// TIA Portal project "Madeta" (V14)

(* hardware
DEVICE "ET 200S station_1"  ET 200S station
   slot 0: "Rack_0"  Rail
   slot 2: "PLC Paletizace pytlu"  IM 151-8 PN/DP CPU  6ES7 151-8AB01-0AB0  V3.2
      slot 1: "PROFINET interface_1"  PN-IO
         slot 1: "Port_1"  Port
         slot 2: "Port_2"  Port
         slot 3: "Port_3"  Port
   slot 4: "PM-E 24VDC_1"  PM-E 24VDC  6ES7 138-4CA01-0AA0
   slot 5: "8DI x 24VDC_1"  8DI x 24VDC  6ES7 131-4BF00-0AA0
   slot 6: "8DI x 24VDC_2"  8DI x 24VDC  6ES7 131-4BF00-0AA0
   slot 7: "8DI x 24VDC_3"  8DI x 24VDC  6ES7 131-4BF00-0AA0
   slot 8: "8DI x 24VDC_4"  8DI x 24VDC  6ES7 131-4BF00-0AA0
   slot 9: "8DI x 24VDC_5"  8DI x 24VDC  6ES7 131-4BF00-0AA0
   slot 10: "8DI x 24VDC_6"  8DI x 24VDC  6ES7 131-4BF00-0AA0
   slot 11: "PM-E 24VDC_2"  PM-E 24VDC  6ES7 138-4CA01-0AA0
   slot 12: "8DO x 24VDC / 0.5A_1"  8DO x 24VDC / 0.5A  6ES7 132-4BF00-0AA0
   slot 13: "PM-E 24VDC_3"  PM-E 24VDC  6ES7 138-4CA01-0AA0
   slot 14: "8DO x 24VDC / 0.5A_2"  8DO x 24VDC / 0.5A  6ES7 132-4BF00-0AA0
   slot 15: "8DO x 24VDC / 0.5A_3"  8DO x 24VDC / 0.5A  6ES7 132-4BF00-0AA0
   slot 16: "8DO x 24VDC / 0.5A_4"  8DO x 24VDC / 0.5A  6ES7 132-4BF00-0AA0
   slot 17: "8DO x 24VDC / 0.5A_5"  8DO x 24VDC / 0.5A  6ES7 132-4BF00-0AA0
DEVICE "GSD device_1"  GSD.Device.PN
   slot 0: "Rack"  Rack  V1.0
   slot 0: "COMAU PAL 180"  X20IF10E3-1  X20IF10E3-1  2.1.x
      slot 0: "DIM 1"  DIM 1
      slot 1: "Interface"  Interface
         slot 1: "Interface - Port1"  Interface - Port1
         slot 2: "Interface - Port2"  Interface - Port2
   slot 1: "8 Bytes In_1"  8 Bytes In
      slot 0: "9"  9
   slot 2: "8 Bytes Out_1"  8 Bytes Out
      slot 0: "10"  10
DEVICE "Panel paletizace pytlu"  KTP600 Basic color PN
   slot 0: "KTP600 Basic color PN"  KTP600 Basic color PN  6AV6 647-0AD11-3AX0  12.0.0.0
   slot 1: "HMI_RT_2"  KTP600 Basic color PN  6AV6 647-0AD11-3AX0  12.0.0.0
   slot 5: "Panel paletizace pytlu.IE_CP_1"  PROFINET Interface  12.0.0.0
      slot 1: "PROFINET Interface_1"  PROFINET Interface
         slot 1: "Port_1"  Port
*)

// ===== PLC "PLC Paletizace pytlu"  IM 151-8 PN/DP CPU =====

VAR_GLOBAL   // PLC tag table "Default tag table"
   "Tag_1" AT %M50.0 : Bool;
   "Manual_Dopravnik_P1" AT %M50.1 : Bool;
   "Manual_Dopravnik_P2_k _oviječce" AT %M50.2 : Bool;
   "Manual_Dopravnik_P3" AT %M50.3 : Bool;
   "Manual_PaletaRovnani_Rozevrit" AT %M60.0 : Bool;
   "Manual_PaletaRovnani_Sevrit" AT %M60.2 : Bool;
   "Manual_Zarazka_P2_Dolu" AT %M60.3 : Bool;
   "Manual_Zarazka_P2_Nahoru" AT %M60.4 : Bool;
   "Manual_Valcovacka" AT %M60.5 : Bool;
   "Automat" AT %M100.0 : Bool;
   "Dopravnik P1 Start" AT %Q6.0 : Bool;
   "Dopravnik P2 do Ovíječky" AT %Q6.1 : Bool;
   "Dopravnik P3 Start" AT %Q6.2 : Bool;
   "Valcovacka Start" AT %Q6.7 : Bool;
   "PaletaRovnani_Rozevrit" AT %Q6.3 : Bool;
   "PaletaRovnani_Sevrit" AT %Q6.4 : Bool;
   "Dopravnik P2 do Stohu" AT %Q6.6 : Bool;
   "Zarazka_P2_Dolu" AT %Q6.5 : Bool;
   "Dveře 2 otevřit" AT %Q7.0 : Bool;
   "Dveře 1 otevřit" AT %Q7.2 : Bool;
   "Dveře 1 otevřeno" AT %Q7.1 : Bool;
   "Dveře 2 otevřeno" AT %Q7.3 : Bool;
   "Dveře 1 požadavek" AT %I3.2 : Bool;
   "Dveře 2 požadavek" AT %I3.5 : Bool;
   "Signální sloupek zelená" AT %Q9.4 : Bool;
   "Tag_2" AT %M150.4 : Bool;
   "Optická závora override" AT %Q10.0 : Bool;
   "Reset" AT %I0.5 : Bool;
   "Override" AT %I0.6 : Bool;
   "Optická závora zapnutí" AT %Q10.1 : Bool;
   "Error" AT %M101.0 : Bool;
   "OP_Start" AT %M90.0 : Bool;
   "OP_Stop" AT %M90.1 : Bool;
   "Tag_3" AT %M200.0 : Bool;
   "Tag_4" AT %M120.0 : Bool;
   "Tag_5" AT %M200.1 : Bool;
   "PřesunP2naOvijecka" AT %M220.0 : Bool;
   "PřesunOvijeckanaP3" AT %M220.1 : Bool;
   "Manual_Oviječka" AT %M50.4 : Bool;
   "Dopravnik Ovijecka Start" AT %Q7.7 : Bool;
   "Manual_Váha" AT %M60.6 : Bool;
   "Pytel na P1" AT %I4.0 : Bool;
   "Rovnání P2 otevřeno" AT %I4.2 : Bool;
   "Paleta P2 u Ovíječky" AT %I4.4 : Bool;
   "Srovnaná paleta na P2" AT %T50 : Timer;
   "Volno na P3" AT %I4.5 : Bool;
   "Ovíječka_Konec balení" AT %I2.5 : Bool;
   "Komunikace robot byte 1" AT %QB256 : Byte;
   "Časovač vypínací impulz váha dopravník" AT %T122 : Timer;
   "Ovíječka_Volná trať" AT %I2.4 : Bool;
   "Ovíječka_Porucha" AT %I2.6 : Bool;
   "Ovíječka_Paleta na točně" AT %I2.7 : Bool;
   "Ovíječce_Start balení" AT %Q9.0 : Bool;
   "Ovíječce_Možno balit" AT %Q9.1 : Bool;
   "Ovíječka_Povolení otevřít dveře" AT %I1.3 : Bool;
   "Manual_RučníPřesunOvnaP3" AT %M50.5 : Bool;
   "Manual_RučníPřesunP2naOv" AT %M50.6 : Bool;
   "Nouzové zastavení" AT %I0.2 : Bool;
   "Tag_6" AT %M200.2 : Bool;
   "Tag_7" AT %T60 : Timer;
   "Pytel na konci Válcovačky" AT %I4.6 : Bool;
   "Časovač volno na váze" AT %T61 : Timer;
   "Tag_9" AT %T62 : Timer;
   "Paleta P2 u stohu" AT %I4.3 : Bool;
   "Manual_Dopravnik_P2_ke_stohu" AT %M50.7 : Bool;
   "Manual_Paletu_P2_ke_stohu" AT %M51.0 : Bool;
   "Manual_Paletu_P2_k_ovíječce" AT %M51.1 : Bool;
   "Časovač_paleta u stohu" AT %T63 : Timer;
   "Časovač_paleta u ovíječky" AT %T64 : Timer;
   "Časovač paleta v ovíječce" AT %T65 : Timer;
   "Timer" AT %T80 : Timer;
   "PHrana I258.4" AT %M80.0 : Bool;
   "Časovač_zapni_pohon_robota" AT %T81 : Timer;
   "Zařízení zapnuto" AT %I0.3 : Bool;
   "Časovač_zapni automat robota" AT %T82 : Timer;
   "Časovač_vypnutí automatu robota" AT %T83 : Timer;
   "Časovač_vypnutí pohonů robota" AT %T84 : Timer;
   "Časovač_spoždění_zapnutí_pohonů robota" AT %T85 : Timer;
   "Časovač_reset alarmů robota" AT %T86 : Timer;
   "Časovač_zpoždění startu" AT %T87 : Timer;
   "Přítomnost palety P2" AT %I4.1 : Bool;
   "Časovač_váha volná" AT %T59 : Timer;
   "Jistič dopravníku P1,P2" AT %I0.1 : Bool;
   "Časovač vadný pytel na váze" AT %T58 : Timer;
   "volný" AT %T123 : Timer;
   "Časovač_start balení" AT %T66 : Timer;
   "Dveře 1 potvrzeno zavření" AT %I3.1 : Bool;
   "Dveře 2 potvrzeno zavření" AT %I3.4 : Bool;
   "Nízký tlak vzduchu" AT %I0.4 : Bool;
   "Jistič válcovačky nebo dopravníku ovíječky" AT %I0.7 : Bool;
   "Porucha kontaktů bezpečnostního relé" AT %I1.0 : Bool;
   "Časovač příliš dlouhý přesun z dopravníku P2" AT %T90 : Timer;
   "Časovač příliš dlouhý přesun z ovíječky" AT %T91 : Timer;
   "Časovač příliš dlouhý přesun palety na dopravníku P2 k ovíječce" AT %T92 : Timer;
   "Časovač píliš dlouhý přesun palety na dopravníku P2 ke stohu" AT %T93 : Timer;
   "Časovač příliš dlouhý chod rovnání palety k paletě" AT %T94 : Timer;
   "Časovač příliš dlouhý chod rovnání palety od palety" AT %T95 : Timer;
   "Světelná závora OK" AT %I1.2 : Bool;
   "Časovač volno na P3" AT %T68 : Timer;
   "Robotovi paleta ve stohu připravena" AT %Q259.0 : Bool;
   "Časovač nová paleta na zmetky" AT %T88 : Timer;
   "Časovač impuls nová paleta na zmetky" AT %T99 : Timer;
   "Signální  sloupek červená" AT %Q9.6 : Bool;
   "Signální sloupek houkačka" AT %Q9.7 : Bool;
   "Signální sloupek oranžová" AT %Q9.5 : Bool;
   "Tag_12" AT %M110.0 : Bool;
   "Tag_13" AT %M110.1 : Bool;
   "Tag_14" AT %M110.2 : Bool;
   "Tag_15" AT %M110.3 : Bool;
   "Tag_8" AT %M150.3 : Bool;
   "Tag_11" AT %M150.0 : Bool;
   "Tag_16" AT %M150.7 : Bool;
   "Tag_17" AT %M150.2 : Bool;
   "Dveře 1 otevřeny" AT %I3.3 : Bool;
   "Tag_18" AT %M40.0 : Bool;
   "Signální sloupek modrá" AT %Q8.7 : Bool;
   "Nouzové zastavení robot neaktivní" AT %I3.6 : Bool;
   "Nouzové zastavení ovíječka neaktivní" AT %I3.7 : Bool;
   "Dveře 2 otevřeny" AT %I3.0 : Bool;
END_VAR

VAR_GLOBAL   // PLC tag table "Errors"
   "Jistič dopravníku P1" AT %I0.0 : Bool;
END_VAR

VAR_GLOBAL   // PLC tag table "Komunikace_robot"
   "Robot_Paletu do pozice stoh" AT %I258.1 : Bool;
   "Robot_paletu do pozice u ovíječky" AT %I258.2 : Bool;
   "Robotovi_P1_Paleta_u_stohu" AT %Q258.0 : Bool;
   "Robotovi_P2_Paleta_u_ovíječky" AT %Q258.1 : Bool;
   "Robotovi_Vadný_pytel" AT %Q258.2 : Bool;
   "Robotovi_Pytel_na_dopravníku" AT %Q258.3 : Bool;
   "Robotovi_polož_novou_paletu" AT %Q258.4 : Bool;
   "Robotovi_paleta_na_zmetky_připravena" AT %Q258.5 : Bool;
   "Robotovi_start_produkce" AT %Q258.6 : Bool;
   "Robotovi_konec_produkce" AT %Q258.7 : Bool;
   "Robotovi_artikl" AT %QB260 : Byte;
   "Robotovi_max_počet_vrstev" AT %QB261 : Byte;
   "Robotovi_aktualní_počet_vrstev" AT %QB262 : Byte;
   "Robotovi_aktualní_počet_pytlů" AT %QB263 : Byte;
   "Robot_potvrzení_zmetku" AT %I258.3 : Bool;
   "Robot_pytel_položen" AT %I258.4 : Bool;
   "Robot_nová_paleta_položena" AT %I258.5 : Bool;
   "Robot_jsem_mimo_dopravník_P1" AT %I258.6 : Bool;
   "Robot_paleta_vadných_polovina" AT %I258.7 : Bool;
   "Robot_paleta_vadných_plná" AT %I259.0 : Bool;
   "Robot_mimo_paletu" AT %I259.1 : Bool;
   "Robot_paleta_plná" AT %I259.2 : Bool;
   "Robot_No alarm" AT %I256.0 : Bool;
   "Robot_Drive on status" AT %I256.1 : Bool;
   "Robot_Start / no hold on mot prog" AT %I256.2 : Bool;
   "Robot_Remote" AT %I256.3 : Bool;
   "Robot_Teach enable (DRI.ON+T1)" AT %I256.4 : Bool;
   "Robot_U1" AT %I256.5 : Bool;
   "Robot_U2" AT %I256.6 : Bool;
   "Robot_U3" AT %I256.7 : Bool;
   "Robot_U4" AT %I257.0 : Bool;
   "Robot_No activa latch alarm" AT %I257.1 : Bool;
   "Robot_Safety speed (for remote)" AT %I257.2 : Bool;
   "Robot_Programing mode" AT %I257.3 : Bool;
   "Robot_State selector in local or remote" AT %I257.5 : Bool;
   "Robot_Systém reddy" AT %I257.6 : Bool;
   "Robot_Heart bit" AT %I257.7 : Bool;
   "Robot_is on HOME" AT %I258.0 : Bool;
   "Robot_reserve" AT %I257.4 : Bool;
   "Robotovi_Drive ON" AT %Q256.0 : Bool;
   "Robotovi_No drive OFF" AT %Q256.1 : Bool;
   "Robotovi_Start" AT %Q256.2 : Bool;
   "Robotovi_No hold" AT %Q256.3 : Bool;
   "Robotovi_U1" AT %Q256.4 : Bool;
   "Robotovi_U2" AT %Q256.5 : Bool;
   "Robotovi_U3" AT %Q256.6 : Bool;
   "Robotovi_U4" AT %Q256.7 : Bool;
   "Robotovi_Cancel alarm" AT %Q257.0 : Bool;
   "Robotovi_Safety speed" AT %Q257.1 : Bool;
   "Robotovi_Reserve" AT %Q257.2 : Bool;
   "Robotovi_Reserve_1" AT %Q257.3 : Bool;
   "Robotovi_Reserve_2" AT %Q257.4 : Bool;
   "Robotovi_Reserve_3" AT %Q257.5 : Bool;
   "Robotovi_Reserve_4" AT %Q257.6 : Bool;
   "Robotovi_Reserve_5" AT %Q257.7 : Bool;
END_VAR

VAR_GLOBAL   // PLC tag table "Komunikace_váha"
   "Váha_Nouzové zastavení" AT %I2.1 : Bool;
   "Váha_Snímač na dopravníku volno" AT %I2.3 : Bool;
   "Dopravník Váha Start" AT %Q8.4 : Bool;
   "Dopravník Váha Stop" AT %Q8.5 : Bool;
   "Váha_motory_zapnuty" AT %I2.0 : Bool;
   "Váha_hmotnost_OK" AT %I2.2 : Bool;
END_VAR

TYPE "Karton"
   STRUCT
      Rotace : Bool;
      Pořadí : Int;
   END_STRUCT;
END_TYPE

// folder: DB

DATA_BLOCK "Komunikace vaha_DB"   // DB3
{ S7_Optimized_Access := 'FALSE' }
VERSION : 0.1
// stored: InstanceOfName Komunikace vaha
"Komunikace vaha"
BEGIN
END_DATA_BLOCK

DATA_BLOCK "Počítadlo_DB"   // DB5
{ S7_Optimized_Access := 'FALSE' }
VERSION : 0.1
// stored: InstanceOfName Počítadlo
"Počítadlo"
BEGIN
END_DATA_BLOCK

DATA_BLOCK "Dopravniky_DB"   // DB10
{ S7_Optimized_Access := 'FALSE' }
VERSION : 0.1
// stored: InstanceOfName Dopravniky
"Dopravniky"
BEGIN
END_DATA_BLOCK

DATA_BLOCK "Klapky_DB"   // DB11
{ S7_Optimized_Access := 'FALSE' }
VERSION : 0.1
// stored: InstanceOfName Klapky
"Klapky"
BEGIN
END_DATA_BLOCK

DATA_BLOCK "Dopravníky pytlů_DB"   // DB12
{ S7_Optimized_Access := 'FALSE' }
VERSION : 0.1
// stored: InstanceOfName Dopravníky pytlů
"Dopravníky pytlů"
BEGIN
END_DATA_BLOCK

DATA_BLOCK "Komunikace robot_DB"   // DB51
{ S7_Optimized_Access := 'FALSE' }
VERSION : 0.1
// stored: InstanceOfName Komunikace robot
"Komunikace robot"
BEGIN
END_DATA_BLOCK

DATA_BLOCK "Komunikace ovijecka_DB"   // DB52
{ S7_Optimized_Access := 'FALSE' }
VERSION : 0.1
// stored: InstanceOfName Komunikace ovijecka
"Komunikace ovijecka"
BEGIN
END_DATA_BLOCK

DATA_BLOCK "Opticka zavora_DB"   // DB54
{ S7_Optimized_Access := 'FALSE' }
VERSION : 0.1
// stored: InstanceOfName Opticka zavora
"Opticka zavora"
BEGIN
END_DATA_BLOCK

DATA_BLOCK "Dvere_DB"   // DB60
{ S7_Optimized_Access := 'FALSE' }
VERSION : 0.1
// stored: InstanceOfName Dvere
"Dvere"
BEGIN
END_DATA_BLOCK

DATA_BLOCK "Signalni sloupek_DB"   // DB61
{ S7_Optimized_Access := 'FALSE' }
VERSION : 0.1
// stored: InstanceOfName Signalni sloupek
"Signalni sloupek"
BEGIN
END_DATA_BLOCK

DATA_BLOCK "Errors_DB"   // DB100
{ S7_Optimized_Access := 'FALSE' }
VERSION : 0.1
// stored: InstanceOfName Errors
"Errors"
BEGIN
END_DATA_BLOCK

DATA_BLOCK "Global_DB"   // DB111
{ S7_Optimized_Access := 'FALSE' }
VERSION : 0.1
// stored: InstanceOfName Global
"Global"
BEGIN
END_DATA_BLOCK

// folder: SystemBlocksFolder/ReportSystemErrorFolder

DATA_BLOCK "RSE_DIAGNOSTIC_STATUS_DB"   // DB127
TITLE = Report System Error Diagnostic Block
{ S7_Optimized_Access := 'FALSE' }
AUTHOR : SIMATIC
FAMILY : RSEDIAG
NAME : RSE7
VERSION : 1.0
// This DB is part of report system error and will be updated by the RSE FB.
//  It is an interface for support of system diagnosis via the CPU web server.
   VAR
      Directory : Struct
         D_Version : Word := WORD#16#0100;   // Version that supports RSE
         D_pGlobalState : Word := WORD#16#0010;   // Byte offset to the start of the "GlobalState" section
         D_pQuery : Word := WORD#16#0014;   // Byte offset to the start of the "Query" section
         D_pComponent : Word := WORD#16#0020;   // Byte offset to the start of the "Component" section
         D_pError : Word := WORD#16#0024;   // Byte offset to the start of the "Error" section
         D_pState : Word := WORD#16#0028;   // Byte offset to the start of the "State" section
         D_pAlarm : Word := WORD#16#005A;   // Byte offset to the start of the "Alarm" section
         D_pSubComponent : Word := WORD#16#0082;   // Byte offset to the start of the "Subcomponent" section
      END_STRUCT;
      GlobalState : Struct
         G_EventCount : Word := WORD#16#0000;   // ID of the last event (counter)
         G_StartReporting : Bool := FALSE;   // Startup evaluation running
      END_STRUCT;
      Query : Struct
         Q_ClientID_User : DWord := DWORD#16#0000_0000;   // ID of the client
         Q_ClientID_Intern : DWord := DWORD#16#0000_0000;   // ID of the client (internal)
         Q_WithSubComponent : Bool := FALSE;   // With/without status of the underlying components (slower)
         Q_SubComponentAlarm : Bool := FALSE;   // AS-iMaster gibt AS-iSlave Alarme zurück
         Q_Reserved2 : Bool := FALSE;   // Reserved
         Q_Reserved3 : Bool := FALSE;   // Reserved
         Q_Reserved4 : Bool := FALSE;   // Reserved
         Q_Reserved5 : Bool := FALSE;   // Reserved
         Q_Reserved6 : Bool := FALSE;   // Reserved
         Q_Reserved7 : Bool := FALSE;   // Reserved
         Q_Start : Bool := FALSE;   // Start query
         Q_Error : Byte := BYTE#16#00;   // Internal error in query
         Q_Reserved8 : Byte := BYTE#16#00;   // Reserved
      END_STRUCT;
      Component : Struct
         C_AddressMode : Byte := BYTE#16#00;   // Addressing mode of the module
         C_Reserved1 : Byte := BYTE#16#00;   // Reserved
         C_ComponentID : Word := WORD#16#0000;   // Hardware ID of the component (internal)
      END_STRUCT;
      Error : Struct
         E_ErrorNo : Word := WORD#16#0000;   // Index of the requested/actual error
         E_LastError : Bool := FALSE;   // TRUE, if E_ErrorNo contains the indes of the last error, otherwise FALSE
      END_STRUCT;
      State : Struct
         S_Hierarchy : Byte := BYTE#16#00;   // Reserved
         S_Periphery : Byte := BYTE#16#00;   // Reserved
         S_SupFault : Bool := FALSE;   // The component is not obtainable
         S_NotAvailable : Bool := FALSE;   // The component does not exist
         S_Faulty : Bool := FALSE;   // The component is disrupted; the "Alarm" section is not empty
         S_MoreErrors : Bool := FALSE;   // There are more errors than RSE can store.
         S_Maintenance1 : Bool := FALSE;   // Maintenance required is indicated
         S_Maintenance2 : Bool := FALSE;   // Maintenance demand is indicated
         S_Deactivated : Bool := FALSE;   // The component was deactivated
         S_Reserved2 : Bool := FALSE;   // Reserved
         S_SubFault : Bool := FALSE;   // An underlying component is disrupted
         S_SubMaintenance1 : Bool := FALSE;   // Maintenance required is indicated for an underlying component
         S_SubMaintenance2 : Bool := FALSE;   // Maintenance demand is indicated for an underlying component
         S_SubDeactivated : Bool := FALSE;   // At least one lower-level component is disabled
         S_Reserved4 : Bool := FALSE;   // Reserved
         S_Reserved5 : Bool := FALSE;   // Reserved
         S_Reserved6 : Bool := FALSE;   // Reserved
         S_Reserved7 : Bool := FALSE;   // Reserved
         S_TIAMS : DWord := DWORD#16#0000_0000;   // Maintenance state of the component
         S_TIAMSChannelExist : DWord := DWORD#16#0000_0000;   // Maintenance state: Configured channels
         S_TIAMSChannelOK : DWord := DWORD#16#0000_0000;   // Maintenance State: Disrupted channels
         S_ChannelCount : Word := WORD#16#0000;   // Number of channels; Valid only when Q_WithSubComponent is set
         S_ChannelVector : Array[0..255] of Bool;   // List of channels involved; Valid only when Q_WithSubComponent is set
      END_STRUCT;
      Alarm : Struct
         A_ComponentID : Word := WORD#16#0000;   // Hardware ID of the component (internal)
         A_TextID1 : Word := WORD#16#0000;   // ID of the first error text
         A_TextLexikonID1 : Word := WORD#16#0000;   // ID of the first error text lexicon
         A_HelpTextLexikonID1 : Word := WORD#16#0000;   // ID of the first help text lexicon
         A_MapTextID : Word := WORD#16#0000;   // ID of the first error text in the export file (HMI)
         A_MapHelpTextID : Word := WORD#16#0000;   // ID of the first help text in the export file (HMI)
         A_TextID2 : Word := WORD#16#0000;   // ID of the second error text
         A_TextLexikonID2 : Word := WORD#16#0000;   // ID of the second error text lexicon
         A_HelpTextLexikonID2 : Word := WORD#16#0000;   // ID of the second help text lexicon
         A_MapTextID2 : Word := WORD#16#0000;   // ID of the second error text in the export file (HMI)
         A_MapHelpTextID2 : Word := WORD#16#0000;   // ID of the second help text in the export file (HMI)
         A_AlarmID : DWord := DWORD#16#0000_0000;   // Message number
         A_ValueCount : Word := WORD#16#000C;   // Number of other occupied bytes
         A_AssociatedValue : Array[1..6] of Word;   // Associated values of the message
      END_STRUCT;
      SubComponent : Struct
         U_SubComponentCount : Word := WORD#16#0000;   // Number of underlying components
         U_SubComponentFault : Array[1..16] of Byte;   // List of status of subordinate components, 1 byte per component
      END_STRUCT;
   END_VAR
BEGIN
END_DATA_BLOCK

// folder: (top level)

ORGANIZATION_BLOCK "Main"   // OB1, LAD
TITLE = "Main Program Sweep (Cycle)"
{ S7_Optimized_Access := 'FALSE' }
VERSION : 0.1
   VAR_TEMP
      OB1_EV_CLASS : Byte;   // Bits 0-3 = 1 (Coming event), Bits 4-7 = 1 (Event class 1)
      OB1_SCAN_1 : Byte;   // 1 (Cold restart scan 1 of OB 1), 3 (Scan 2-n of OB 1)
      OB1_PRIORITY : Byte;   // Priority of OB Execution
      OB1_OB_NUMBR : Byte;   // 1 (Organization block 1, OB1)
      OB1_RESERVED_1 : Byte;   // Reserved for system
      OB1_RESERVED_2 : Byte;   // Reserved for system
      OB1_PREV_CYCLE : Int;   // Cycle time of previous OB1 scan (milliseconds)
      OB1_MIN_CYCLE : Int;   // Minimum cycle time of OB1 (milliseconds)
      OB1_MAX_CYCLE : Int;   // Maximum cycle time of OB1 (milliseconds)
      OB1_DATE_TIME : Date_And_Time;   // Date and time OB1 started
   END_VAR
BEGIN

REGION Network 1
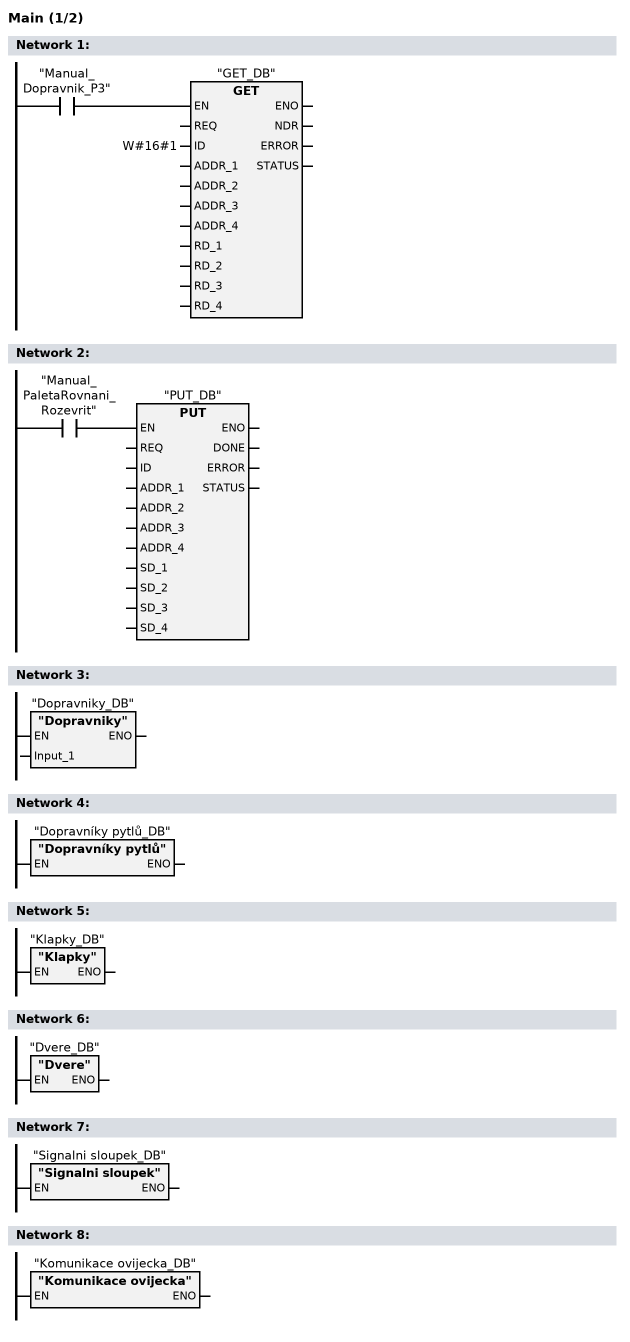
   IF "Manual_Dopravnik_P3" THEN
       "GET_DB"(ID := W#16#1);   // GET
   END_IF;
END_REGION

REGION Network 2
   IF "Manual_PaletaRovnani_Rozevrit" THEN
       "PUT_DB"();   // PUT
   END_IF;
END_REGION

REGION Network 3
   RUNG wire#powerrail
      "Dopravniky_DB"(Input_1 :=)
   END_RUNG
   // the same network as SCL:
   "Dopravniky_DB"();   // "Dopravniky"
END_REGION

REGION Network 4
   RUNG wire#powerrail
      "Dopravníky pytlů_DB"()
   END_RUNG
   // the same network as SCL:
   "Dopravníky pytlů_DB"();   // "Dopravníky pytlů"
END_REGION

REGION Network 5
   RUNG wire#powerrail
      "Klapky_DB"()
   END_RUNG
   // the same network as SCL:
   "Klapky_DB"();   // "Klapky"
END_REGION

REGION Network 6
   RUNG wire#powerrail
      "Dvere_DB"()
   END_RUNG
   // the same network as SCL:
   "Dvere_DB"();   // "Dvere"
END_REGION

REGION Network 7
   RUNG wire#powerrail
      "Signalni sloupek_DB"()
   END_RUNG
   // the same network as SCL:
   "Signalni sloupek_DB"();   // "Signalni sloupek"
END_REGION

REGION Network 8
   RUNG wire#powerrail
      "Komunikace ovijecka_DB"()
   END_RUNG
   // the same network as SCL:
   "Komunikace ovijecka_DB"();   // "Komunikace ovijecka"
END_REGION

REGION Network 9
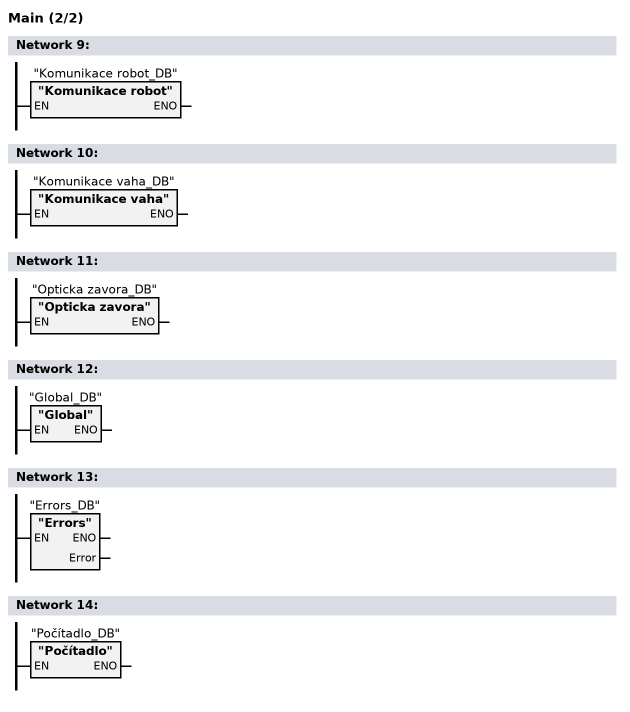
   RUNG wire#powerrail
      "Komunikace robot_DB"()
   END_RUNG
   // the same network as SCL:
   "Komunikace robot_DB"();   // "Komunikace robot"
END_REGION

REGION Network 10
   RUNG wire#powerrail
      "Komunikace vaha_DB"()
   END_RUNG
   // the same network as SCL:
   "Komunikace vaha_DB"();   // "Komunikace vaha"
END_REGION

REGION Network 11
   RUNG wire#powerrail
      "Opticka zavora_DB"()
   END_RUNG
   // the same network as SCL:
   "Opticka zavora_DB"();   // "Opticka zavora"
END_REGION

REGION Network 12
   RUNG wire#powerrail
      "Global_DB"()
   END_RUNG
   // the same network as SCL:
   "Global_DB"();   // "Global"
END_REGION

REGION Network 13
   RUNG wire#powerrail
      "Errors_DB"(Error =>)
   END_RUNG
   // the same network as SCL:
   "Errors_DB"();   // "Errors"
END_REGION

REGION Network 14
   RUNG wire#powerrail
      "Počítadlo_DB"()
   END_RUNG
   // the same network as SCL:
   "Počítadlo_DB"();   // "Počítadlo"
END_REGION

REGION Network 16 (STL): Call system diagnostics block
         CALL  "RSE_FB", "RSE_DB";
END_REGION
END_ORGANIZATION_BLOCK

ORGANIZATION_BLOCK "OB80"   // OB80, LAD
{ S7_Optimized_Access := 'FALSE' }
VERSION : 0.1
   VAR_TEMP
      Temp_0 : Byte;
      Temp_1 : Byte;
      Temp_2 : Byte;
      Temp_3 : Byte;
      Temp_4 : Byte;
      Temp_5 : Byte;
      Temp_6 : Word;
      Temp_7 : Byte;
      Temp_8 : Byte;
      Temp_9 : Byte;
      Temp_10 : Byte;
      Temp_11 : Date_And_Time;
   END_VAR
BEGIN
END_ORGANIZATION_BLOCK

ORGANIZATION_BLOCK "OB82"   // OB82, LAD
{ S7_Optimized_Access := 'FALSE' }
VERSION : 0.1
   VAR_TEMP
      Temp_0 : Byte;
      Temp_1 : Byte;
      Temp_2 : Byte;
      Temp_3 : Byte;
      Temp_4 : Byte;
      Temp_5 : Byte;
      Temp_6 : Word;
      Temp_7 : Bool;
      Temp_8 : Bool;
      Temp_9 : Bool;
      Temp_10 : Bool;
      Temp_11 : Bool;
      Temp_12 : Bool;
      Temp_13 : Bool;
      Temp_14 : Bool;
      Temp_15 : Byte;
      Temp_16 : Bool;
      Temp_17 : Bool;
      Temp_18 : Bool;
      Temp_19 : Bool;
      Temp_20 : Bool;
      Temp_21 : Bool;
      Temp_22 : Bool;
      Temp_23 : Bool;
      Temp_24 : Bool;
      Temp_25 : Bool;
      Temp_26 : Bool;
      Temp_27 : Bool;
      Temp_28 : Bool;
      Temp_29 : Bool;
      Temp_30 : Bool;
      Temp_31 : Bool;
      Temp_32 : Date_And_Time;
   END_VAR
BEGIN

REGION Network 1 (STL): Call system diagnostics block
         CALL  "RSE_FB", "RSE_DB";
END_REGION
END_ORGANIZATION_BLOCK

ORGANIZATION_BLOCK "OB83"   // OB83, LAD
{ S7_Optimized_Access := 'FALSE' }
VERSION : 0.1
   VAR_TEMP
      Temp_0 : Byte;
      Temp_1 : Byte;
      Temp_2 : Byte;
      Temp_3 : Byte;
      Temp_4 : Byte;
      Temp_5 : Byte;
      Temp_6 : Word;
      Temp_7 : Int;
      Temp_8 : Word;
      Temp_9 : Date_And_Time;
   END_VAR
BEGIN

REGION Network 1 (STL): Call system diagnostics block
         CALL  "RSE_FB", "RSE_DB";
END_REGION
END_ORGANIZATION_BLOCK

ORGANIZATION_BLOCK "OB85"   // OB85, LAD
{ S7_Optimized_Access := 'FALSE' }
VERSION : 0.1
   VAR_TEMP
      Temp_0 : Byte;
      Temp_1 : Byte;
      Temp_2 : Byte;
      Temp_3 : Byte;
      Temp_4 : Byte;
      Temp_5 : Byte;
      Temp_6 : Int;
      Temp_7 : Byte;
      Temp_8 : Byte;
      Temp_9 : Byte;
      Temp_10 : Byte;
      Temp_11 : Date_And_Time;
   END_VAR
BEGIN
END_ORGANIZATION_BLOCK

ORGANIZATION_BLOCK "OB86"   // OB86, LAD
{ S7_Optimized_Access := 'FALSE' }
VERSION : 0.1
   VAR_TEMP
      Temp_0 : Byte;
      Temp_1 : Byte;
      Temp_2 : Byte;
      Temp_3 : Byte;
      Temp_4 : Byte;
      Temp_5 : Byte;
      Temp_6 : Word;
      Temp_7 : Array[0..31] of Bool;
      Temp_8 : Date_And_Time;
   END_VAR
BEGIN

REGION Network 1 (STL): Call system diagnostics block
         CALL  "RSE_FB", "RSE_DB";
END_REGION
END_ORGANIZATION_BLOCK

ORGANIZATION_BLOCK "OB87"   // OB87, LAD
{ S7_Optimized_Access := 'FALSE' }
VERSION : 0.1
   VAR_TEMP
      Temp_0 : Byte;
      Temp_1 : Byte;
      Temp_2 : Byte;
      Temp_3 : Byte;
      Temp_4 : Byte;
      Temp_5 : Byte;
      Temp_6 : Word;
      Temp_7 : DWord;
      Temp_8 : Date_And_Time;
   END_VAR
BEGIN
END_ORGANIZATION_BLOCK

ORGANIZATION_BLOCK "OB100"   // OB100, LAD
{ S7_Optimized_Access := 'FALSE' }
VERSION : 0.1
   VAR_TEMP
      Temp_0 : Byte;
      Temp_1 : Byte;
      Temp_2 : Byte;
      Temp_3 : Byte;
      Temp_4 : Byte;
      Temp_5 : Byte;
      Temp_6 : Word;
      Temp_7 : DWord;
      Temp_8 : Date_And_Time;
   END_VAR
BEGIN
END_ORGANIZATION_BLOCK

ORGANIZATION_BLOCK "OB121"   // OB121, LAD
{ S7_Optimized_Access := 'FALSE' }
VERSION : 0.1
   VAR_TEMP
      Temp_0 : Byte;
      Temp_1 : Byte;
      Temp_2 : Byte;
      Temp_3 : Byte;
      Temp_4 : Byte;
      Temp_5 : Byte;
      Temp_6 : Word;
      Temp_7 : Word;
      Temp_8 : Word;
      Temp_9 : Date_And_Time;
   END_VAR
BEGIN
END_ORGANIZATION_BLOCK

ORGANIZATION_BLOCK "OB122"   // OB122, LAD
{ S7_Optimized_Access := 'FALSE' }
VERSION : 0.1
   VAR_TEMP
      Temp_0 : Byte;
      Temp_1 : Byte;
      Temp_2 : Byte;
      Temp_3 : Byte;
      Temp_4 : Byte;
      Temp_5 : Byte;
      Temp_6 : Word;
      Temp_7 : Word;
      Temp_8 : Word;
      Temp_9 : Date_And_Time;
   END_VAR
BEGIN
END_ORGANIZATION_BLOCK

// folder: Function Block

FUNCTION_BLOCK "Global"   // FB1, LAD
{ S7_Optimized_Access := 'FALSE' }
VERSION : 0.1
   VAR_TEMP
      Start : Bool;
      Stop : Bool;
   END_VAR
   VAR_TEMP   // added for the SCL form of the ladder/FBD networks
      _w1 : Bool;
   END_VAR
BEGIN

REGION Network 1
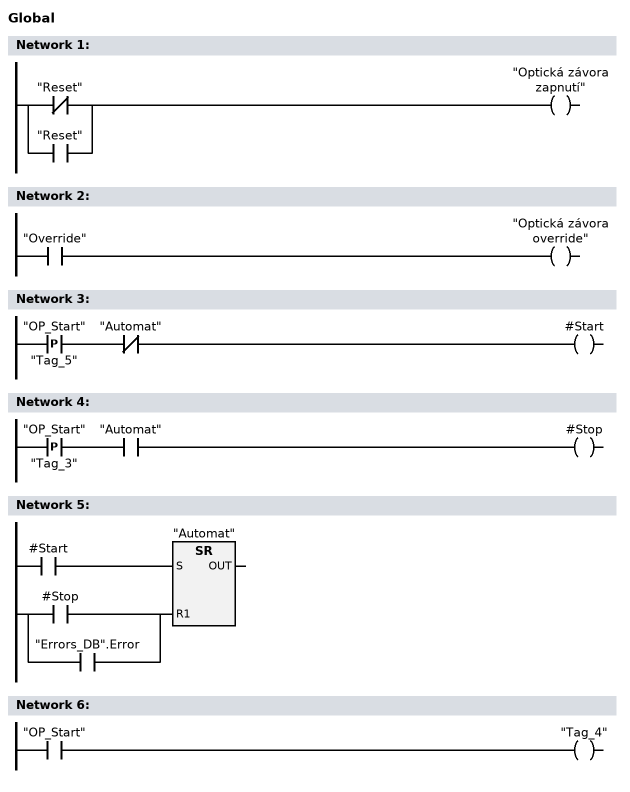
   RUNG wire#powerrail
      I_Contact( "Reset" )
      wire#w1
      Coil( "Optická závora zapnutí" )
   END_RUNG
   RUNG wire#powerrail
      Contact( "Reset" )
   END_RUNG wire#w1
   // the same network as SCL:
   "Optická závora zapnutí" := NOT "Reset" OR "Reset";
END_REGION

REGION Network 2
   RUNG wire#powerrail
      Contact( "Override" )
      Coil( "Optická závora override" )
   END_RUNG
   // the same network as SCL:
   "Optická závora override" := "Override";
END_REGION

REGION Network 3
   RUNG wire#powerrail
      P_Contact(operand := "OP_Start", bit := "Tag_5")
      I_Contact( "Automat" )
      Coil( #Start )
   END_RUNG
   // the same network as SCL:
   #_w1 := "OP_Start" AND NOT "Tag_5";   // rising edge of "OP_Start"
   "Tag_5" := "OP_Start";
   #Start := #_w1 AND NOT "Automat";
END_REGION

REGION Network 4
   RUNG wire#powerrail
      P_Contact(operand := "OP_Start", bit := "Tag_3")
      Contact( "Automat" )
      Coil( #Stop )
   END_RUNG
   // the same network as SCL:
   #_w1 := "OP_Start" AND NOT "Tag_3";   // rising edge of "OP_Start"
   "Tag_3" := "OP_Start";
   #Stop := #_w1 AND "Automat";
END_REGION

REGION Network 5
   RUNG wire#powerrail
      Contact( #Start )
      S_SR(operand := "Automat", r1 := wire#w1)
   END_RUNG
   RUNG wire#powerrail
      Contact( #Stop )
   END_RUNG wire#w1
   RUNG wire#powerrail
      Contact( "Errors_DB".Error )
   END_RUNG wire#w1
   // the same network as SCL:
   IF #Start THEN
       "Automat" := TRUE;   // SR flip-flop
   END_IF;
   IF #Stop OR "Errors_DB".Error THEN "Automat" := FALSE; END_IF;
END_REGION

REGION Network 6
   RUNG wire#powerrail
      Contact( "OP_Start" )
      Coil( "Tag_4" )
   END_RUNG
   // the same network as SCL:
   "Tag_4" := "OP_Start";
END_REGION
END_FUNCTION_BLOCK

FUNCTION_BLOCK "Počítadlo"   // FB4, LAD
{ S7_Optimized_Access := 'FALSE' }
VERSION : 0.1
   VAR
      ČísloArtiklu : Int;
      "Maximální počet vrstev" : Int := 12;
      "Počet Vrstev" : Int;
      "Aktuální počet vrstev" : Int;
      "Aktuální počet pytlů" : Int;
      "Min počet vrstev ovíjení" : Int;
   END_VAR
   VAR_TEMP
      pocetpytlůPlus1 : Int;
   END_VAR
   VAR_TEMP   // added for the SCL form of the ladder/FBD networks
      _w1 : Bool;
   END_VAR
BEGIN

REGION Network 1
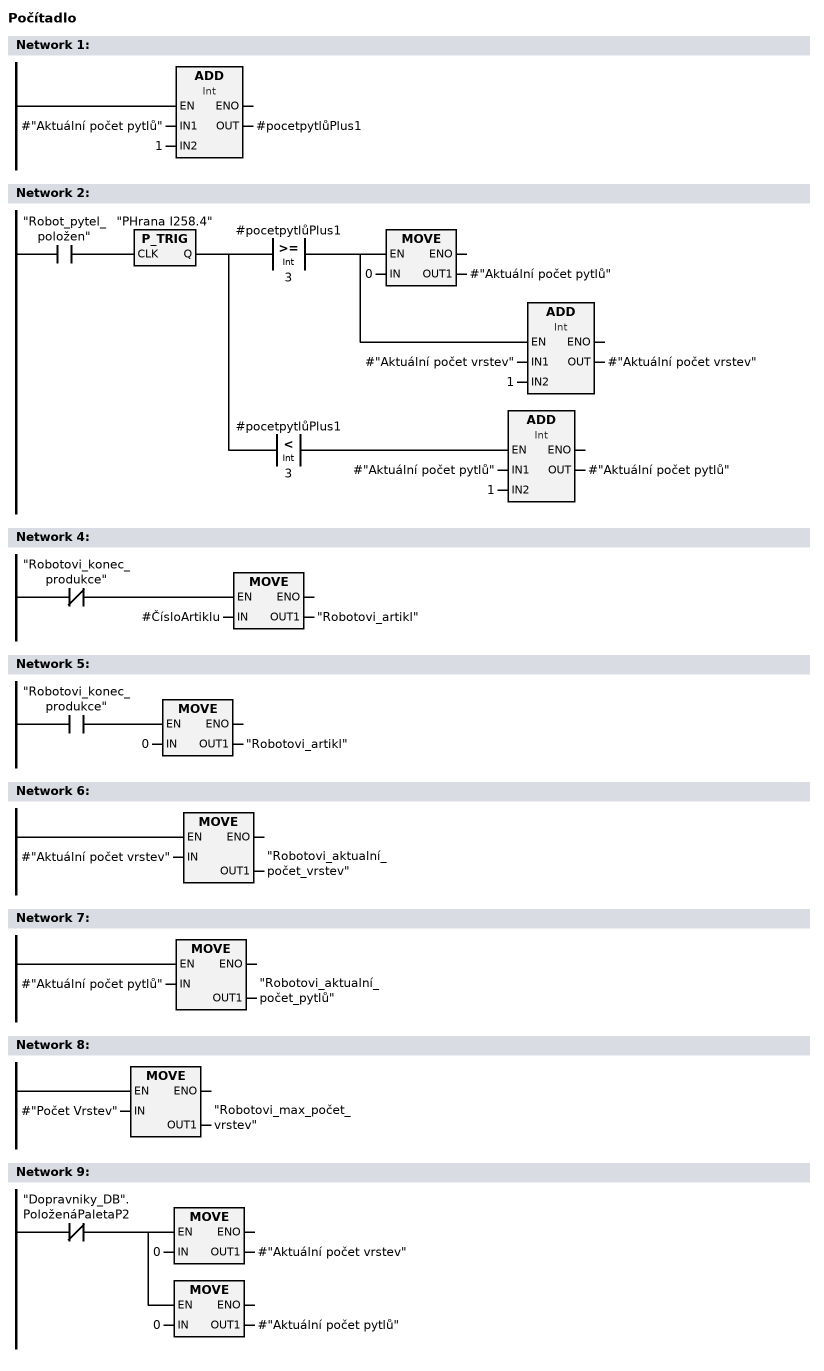
   RUNG wire#powerrail
      { S7_Templates := "SrcType := Int"; S7_GenerateENO := "TRUE" } Add(in1 := #"Aktuální počet pytlů", in2 := 1, out => #pocetpytlůPlus1)
   END_RUNG
   // the same network as SCL:
   #pocetpytlůPlus1 := #"Aktuální počet pytlů" + 1;
END_REGION

REGION Network 2
   RUNG wire#powerrail
      Contact( "Robot_pytel_položen" )
      P_Trig( "PHrana I258.4" )
      wire#w1
      { S7_Templates := "SrcType := Int" } GE_Contact(in1 := #pocetpytlůPlus1, in2 := 3)
      wire#w2
      { S7_GenerateENO := "TRUE" } Move(in := 0, out1 => #"Aktuální počet pytlů")
   END_RUNG
   RUNG wire#w2
      { S7_Templates := "SrcType := Int"; S7_GenerateENO := "TRUE" } Add(in1 := #"Aktuální počet vrstev", in2 := 1, out => #"Aktuální počet vrstev")
   END_RUNG
   RUNG wire#w1
      { S7_Templates := "SrcType := Int" } LT_Contact(in1 := #pocetpytlůPlus1, in2 := 3)
      { S7_Templates := "SrcType := Int"; S7_GenerateENO := "TRUE" } Add(in1 := #"Aktuální počet pytlů", in2 := 1, out => #"Aktuální počet pytlů")
   END_RUNG
   // the same network as SCL:
   #_w1 := "Robot_pytel_položen" AND NOT "PHrana I258.4";   // rising edge
   "PHrana I258.4" := "Robot_pytel_položen";
   IF #_w1 AND (#pocetpytlůPlus1 >= 3) THEN
       #"Aktuální počet pytlů" := 0;
       #"Aktuální počet vrstev" := #"Aktuální počet vrstev" + 1;
   END_IF;
   IF #_w1 AND (#pocetpytlůPlus1 < 3) THEN #"Aktuální počet pytlů" := #"Aktuální počet pytlů" + 1; END_IF;
END_REGION

REGION Network 4
   RUNG wire#powerrail
      I_Contact( "Robotovi_konec_produkce" )
      { S7_GenerateENO := "TRUE" } Move(in := #ČísloArtiklu, out1 => "Robotovi_artikl")
   END_RUNG
   // the same network as SCL:
   IF NOT "Robotovi_konec_produkce" THEN "Robotovi_artikl" := #ČísloArtiklu; END_IF;
END_REGION

REGION Network 5
   RUNG wire#powerrail
      Contact( "Robotovi_konec_produkce" )
      { S7_GenerateENO := "TRUE" } Move(in := 0, out1 => "Robotovi_artikl")
   END_RUNG
   // the same network as SCL:
   IF "Robotovi_konec_produkce" THEN "Robotovi_artikl" := 0; END_IF;
END_REGION

REGION Network 6
   RUNG wire#powerrail
      { S7_GenerateENO := "TRUE" } Move(in := #"Aktuální počet vrstev", out1 => "Robotovi_aktualní_počet_vrstev")
   END_RUNG
   // the same network as SCL:
   "Robotovi_aktualní_počet_vrstev" := #"Aktuální počet vrstev";
END_REGION

REGION Network 7
   RUNG wire#powerrail
      { S7_GenerateENO := "TRUE" } Move(in := #"Aktuální počet pytlů", out1 => "Robotovi_aktualní_počet_pytlů")
   END_RUNG
   // the same network as SCL:
   "Robotovi_aktualní_počet_pytlů" := #"Aktuální počet pytlů";
END_REGION

REGION Network 8
   RUNG wire#powerrail
      { S7_GenerateENO := "TRUE" } Move(in := #"Počet Vrstev", out1 => "Robotovi_max_počet_vrstev")
   END_RUNG
   // the same network as SCL:
   "Robotovi_max_počet_vrstev" := #"Počet Vrstev";
END_REGION

REGION Network 9
   RUNG wire#powerrail
      I_Contact( "Dopravniky_DB".PoloženáPaletaP2 )
      wire#w1
      { S7_GenerateENO := "TRUE" } Move(in := 0, out1 => #"Aktuální počet vrstev")
   END_RUNG
   RUNG wire#w1
      { S7_GenerateENO := "TRUE" } Move(in := 0, out1 => #"Aktuální počet pytlů")
   END_RUNG
   // the same network as SCL:
   IF NOT "Dopravniky_DB".PoloženáPaletaP2 THEN
       #"Aktuální počet vrstev" := 0;
       #"Aktuální počet pytlů" := 0;
   END_IF;
END_REGION
END_FUNCTION_BLOCK

FUNCTION_BLOCK "Dopravniky"   // FB10, LAD
TITLE = Dopravniky
{ S7_Optimized_Access := 'FALSE' }
VERSION : 0.1
   VAR_INPUT
      Input_1 : Block_FB;
   END_VAR
   VAR
      PřesunP2naOvijecka : Bool;
      PoloženáPaletaP2 : Bool;
      SrovnanáPaletaP2 : Bool;
      PřesunOvijeckaNaP3 : Bool;
      "Paleta u ovíječky" : Bool;
      "Paleta u stohu" : Bool;
      "Paleta na točně" : Bool;
      "Ovinutá paleta" : Bool;
      "Nebalit paletu na P2" : Bool;
      "Nebalit paletu na Ovíječce" : Bool;
   END_VAR
   VAR_TEMP   // added for the SCL form of the ladder/FBD networks
      _w1 : Bool;
      _s5time1 : S5Time;
   END_VAR
BEGIN

REGION Network 1
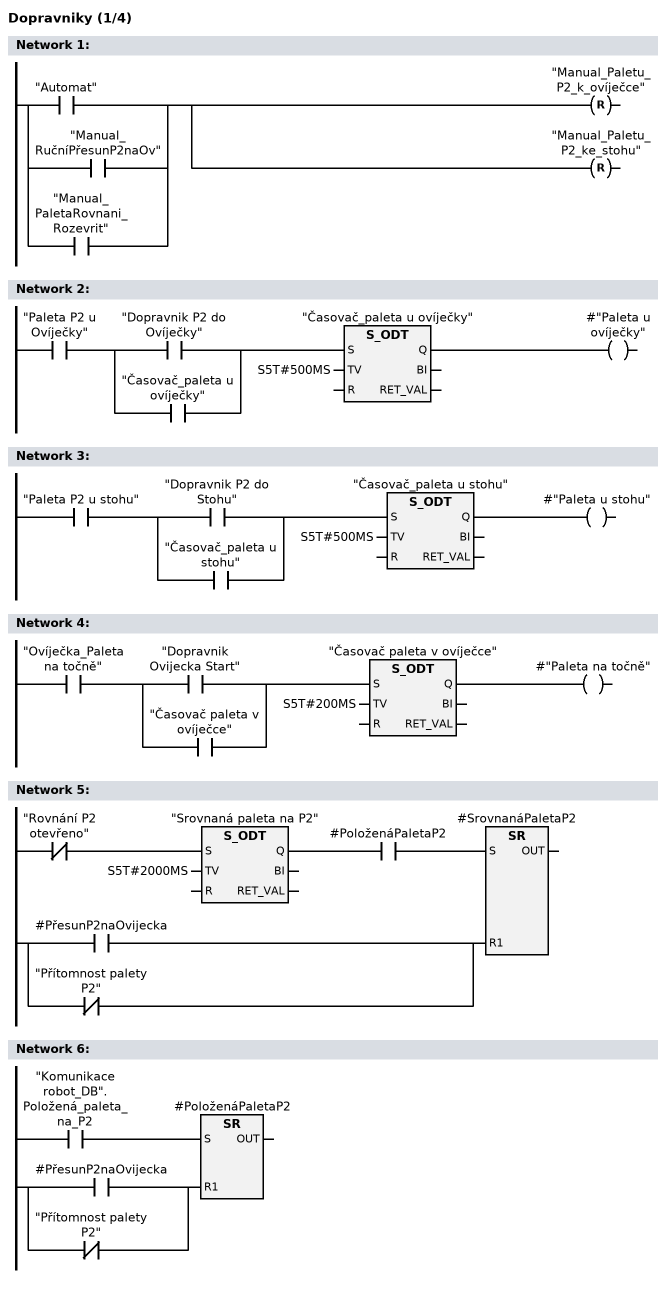
   RUNG wire#powerrail
      Contact( "Automat" )
      wire#w1
      R_Coil( "Manual_Paletu_P2_k_ovíječce" )
   END_RUNG
   RUNG wire#powerrail
      Contact( "Manual_RučníPřesunP2naOv" )
   END_RUNG wire#w1
   RUNG wire#powerrail
      Contact( "Manual_PaletaRovnani_Rozevrit" )
   END_RUNG wire#w1
   RUNG wire#w1
      R_Coil( "Manual_Paletu_P2_ke_stohu" )
   END_RUNG
   // the same network as SCL:
   IF "Automat" OR "Manual_RučníPřesunP2naOv" OR "Manual_PaletaRovnani_Rozevrit" THEN
       "Manual_Paletu_P2_k_ovíječce" := FALSE;
       "Manual_Paletu_P2_ke_stohu" := FALSE;
   END_IF;
END_REGION

REGION Network 2
   RUNG wire#powerrail
      Contact( "Paleta P2 u Ovíječky" )
      wire#w1
      Contact( "Dopravnik P2 do Ovíječky" )
      wire#w2
      S_ODT(T_NO := "Časovač_paleta u ovíječky", TV := S5T#500MS, R :=, BI =>, RET_VAL =>)
      Coil( #"Paleta u ovíječky" )
   END_RUNG
   RUNG wire#w1
      Contact( "Časovač_paleta u ovíječky" )
   END_RUNG wire#w2
   // the same network as SCL:
   #_s5time1 := S_ODT(T_NO := "Časovač_paleta u ovíječky",
                      S := "Paleta P2 u Ovíječky" AND ("Dopravnik P2 do Ovíječky" OR "Časovač_paleta u ovíječky"),
                      TV := S5T#500MS,
                      Q => #_w1);
   #"Paleta u ovíječky" := #_w1;
END_REGION

REGION Network 3
   RUNG wire#powerrail
      Contact( "Paleta P2 u stohu" )
      wire#w1
      Contact( "Dopravnik P2 do Stohu" )
      wire#w2
      S_ODT(T_NO := "Časovač_paleta u stohu", TV := S5T#500MS, R :=, BI =>, RET_VAL =>)
      Coil( #"Paleta u stohu" )
   END_RUNG
   RUNG wire#w1
      Contact( "Časovač_paleta u stohu" )
   END_RUNG wire#w2
   // the same network as SCL:
   #_s5time1 := S_ODT(T_NO := "Časovač_paleta u stohu",
                      S := "Paleta P2 u stohu" AND ("Dopravnik P2 do Stohu" OR "Časovač_paleta u stohu"),
                      TV := S5T#500MS,
                      Q => #_w1);
   #"Paleta u stohu" := #_w1;
END_REGION

REGION Network 4
   RUNG wire#powerrail
      Contact( "Ovíječka_Paleta na točně" )
      wire#w1
      Contact( "Dopravnik Ovijecka Start" )
      wire#w2
      S_ODT(T_NO := "Časovač paleta v ovíječce", TV := S5T#200MS, R :=, BI =>, RET_VAL =>)
      Coil( #"Paleta na točně" )
   END_RUNG
   RUNG wire#w1
      Contact( "Časovač paleta v ovíječce" )
   END_RUNG wire#w2
   // the same network as SCL:
   #_s5time1 := S_ODT(T_NO := "Časovač paleta v ovíječce",
                      S := "Ovíječka_Paleta na točně" AND ("Dopravnik Ovijecka Start" OR "Časovač paleta v ovíječce"),
                      TV := S5T#200MS,
                      Q => #_w1);
   #"Paleta na točně" := #_w1;
END_REGION

REGION Network 5
   RUNG wire#powerrail
      I_Contact( "Rovnání P2 otevřeno" )
      S_ODT(T_NO := "Srovnaná paleta na P2", TV := S5T#2000MS, R :=, BI =>, RET_VAL =>)
      Contact( #PoloženáPaletaP2 )
      S_SR(operand := #SrovnanáPaletaP2, r1 := wire#w1)
   END_RUNG
   RUNG wire#powerrail
      Contact( #PřesunP2naOvijecka )
   END_RUNG wire#w1
   RUNG wire#powerrail
      I_Contact( "Přítomnost palety P2" )
   END_RUNG wire#w1
   // the same network as SCL:
   #_s5time1 := S_ODT(T_NO := "Srovnaná paleta na P2",
                      S := NOT "Rovnání P2 otevřeno",
                      TV := S5T#2000MS,
                      Q => #_w1);
   IF #_w1 AND #PoloženáPaletaP2 THEN
       #SrovnanáPaletaP2 := TRUE;   // SR flip-flop
   END_IF;
   IF #PřesunP2naOvijecka OR NOT "Přítomnost palety P2" THEN #SrovnanáPaletaP2 := FALSE; END_IF;
END_REGION

REGION Network 6
   RUNG wire#powerrail
      Contact( "Komunikace robot_DB".Položená_paleta_na_P2 )
      S_SR(operand := #PoloženáPaletaP2, r1 := wire#w1)
   END_RUNG
   RUNG wire#powerrail
      Contact( #PřesunP2naOvijecka )
   END_RUNG wire#w1
   RUNG wire#powerrail
      I_Contact( "Přítomnost palety P2" )
   END_RUNG wire#w1
   // the same network as SCL:
   IF "Komunikace robot_DB".Položená_paleta_na_P2 THEN
       #PoloženáPaletaP2 := TRUE;   // SR flip-flop
   END_IF;
   IF #PřesunP2naOvijecka OR NOT "Přítomnost palety P2" THEN #PoloženáPaletaP2 := FALSE; END_IF;
END_REGION

REGION Network 7
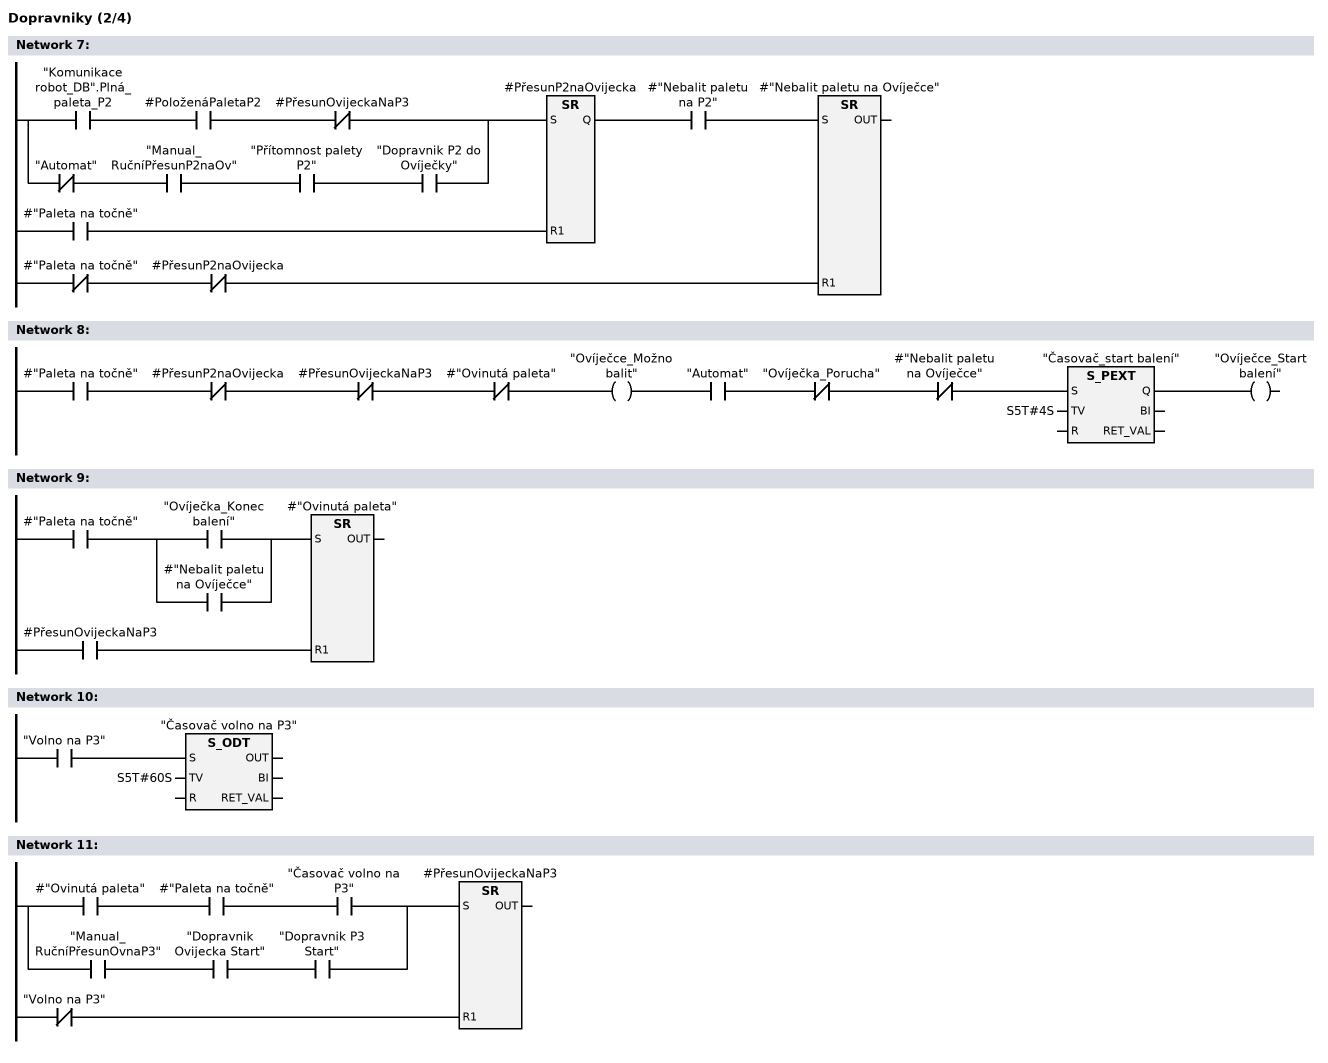
   RUNG wire#powerrail
      Contact( "Komunikace robot_DB".Plná_paleta_P2 )
      Contact( #PoloženáPaletaP2 )
      I_Contact( #PřesunOvijeckaNaP3 )
      wire#w1
      S_SR(operand := #PřesunP2naOvijecka, r1 := wire#w2)
      Contact( #"Nebalit paletu na P2" )
      S_SR(operand := #"Nebalit paletu na Ovíječce", r1 := wire#w3)
   END_RUNG
   RUNG wire#powerrail
      I_Contact( "Automat" )
      Contact( "Manual_RučníPřesunP2naOv" )
      Contact( "Přítomnost palety P2" )
      Contact( "Dopravnik P2 do Ovíječky" )
   END_RUNG wire#w1
   RUNG wire#powerrail
      Contact( #"Paleta na točně" )
   END_RUNG wire#w2
   RUNG wire#powerrail
      I_Contact( #"Paleta na točně" )
      I_Contact( #PřesunP2naOvijecka )
   END_RUNG wire#w3
   // the same network as SCL:
   IF ("Komunikace robot_DB".Plná_paleta_P2 AND #PoloženáPaletaP2 AND NOT #PřesunOvijeckaNaP3) OR (NOT "Automat" AND "Manual_RučníPřesunP2naOv" AND "Přítomnost palety P2" AND "Dopravnik P2 do Ovíječky") THEN
       #PřesunP2naOvijecka := TRUE;   // SR flip-flop
   END_IF;
   IF #"Paleta na točně" THEN #PřesunP2naOvijecka := FALSE; END_IF;
   IF #PřesunP2naOvijecka AND #"Nebalit paletu na P2" THEN
       #"Nebalit paletu na Ovíječce" := TRUE;   // SR flip-flop
   END_IF;
   IF NOT #"Paleta na točně" AND NOT #PřesunP2naOvijecka THEN #"Nebalit paletu na Ovíječce" := FALSE; END_IF;
END_REGION

REGION Network 8
   RUNG wire#powerrail
      Contact( #"Paleta na točně" )
      I_Contact( #PřesunP2naOvijecka )
      I_Contact( #PřesunOvijeckaNaP3 )
      I_Contact( #"Ovinutá paleta" )
      Coil( "Ovíječce_Možno balit" )
      Contact( "Automat" )
      I_Contact( "Ovíječka_Porucha" )
      I_Contact( #"Nebalit paletu na Ovíječce" )
      S_PEXT(T_NO := "Časovač_start balení", TV := S5T#4S, R :=, BI =>, RET_VAL =>)
      Coil( "Ovíječce_Start balení" )
   END_RUNG
   // the same network as SCL:
   "Ovíječce_Možno balit" := #"Paleta na točně" AND NOT #PřesunP2naOvijecka AND NOT #PřesunOvijeckaNaP3 AND NOT #"Ovinutá paleta";
   #_s5time1 := S_PEXT(T_NO := "Časovač_start balení",
                       S := "Ovíječce_Možno balit" AND "Automat" AND NOT "Ovíječka_Porucha" AND NOT #"Nebalit paletu na Ovíječce",
                       TV := S5T#4S,
                       Q => #_w1);
   "Ovíječce_Start balení" := #_w1;
END_REGION

REGION Network 9
   RUNG wire#powerrail
      Contact( #"Paleta na točně" )
      wire#w1
      Contact( "Ovíječka_Konec balení" )
      wire#w2
      S_SR(operand := #"Ovinutá paleta", r1 := wire#w3)
   END_RUNG
   RUNG wire#w1
      Contact( #"Nebalit paletu na Ovíječce" )
   END_RUNG wire#w2
   RUNG wire#powerrail
      Contact( #PřesunOvijeckaNaP3 )
   END_RUNG wire#w3
   // the same network as SCL:
   IF #"Paleta na točně" AND ("Ovíječka_Konec balení" OR #"Nebalit paletu na Ovíječce") THEN
       #"Ovinutá paleta" := TRUE;   // SR flip-flop
   END_IF;
   IF #PřesunOvijeckaNaP3 THEN #"Ovinutá paleta" := FALSE; END_IF;
END_REGION

REGION Network 10
   RUNG wire#powerrail
      Contact( "Volno na P3" )
      S_ODT(T_NO := "Časovač volno na P3", TV := S5T#60S, R :=, BI =>, RET_VAL =>)
   END_RUNG
   // the same network as SCL:
   #_s5time1 := S_ODT(T_NO := "Časovač volno na P3", S := "Volno na P3", TV := S5T#60S);
END_REGION

REGION Network 11
   RUNG wire#powerrail
      Contact( #"Ovinutá paleta" )
      Contact( #"Paleta na točně" )
      Contact( "Časovač volno na P3" )
      wire#w1
      S_SR(operand := #PřesunOvijeckaNaP3, r1 := wire#w2)
   END_RUNG
   RUNG wire#powerrail
      Contact( "Manual_RučníPřesunOvnaP3" )
      Contact( "Dopravnik Ovijecka Start" )
      Contact( "Dopravnik P3 Start" )
   END_RUNG wire#w1
   RUNG wire#powerrail
      I_Contact( "Volno na P3" )
   END_RUNG wire#w2
   // the same network as SCL:
   IF (#"Ovinutá paleta" AND #"Paleta na točně" AND "Časovač volno na P3") OR ("Manual_RučníPřesunOvnaP3" AND "Dopravnik Ovijecka Start" AND "Dopravnik P3 Start") THEN
       #PřesunOvijeckaNaP3 := TRUE;   // SR flip-flop
   END_IF;
   IF NOT "Volno na P3" THEN #PřesunOvijeckaNaP3 := FALSE; END_IF;
END_REGION

REGION Network 12
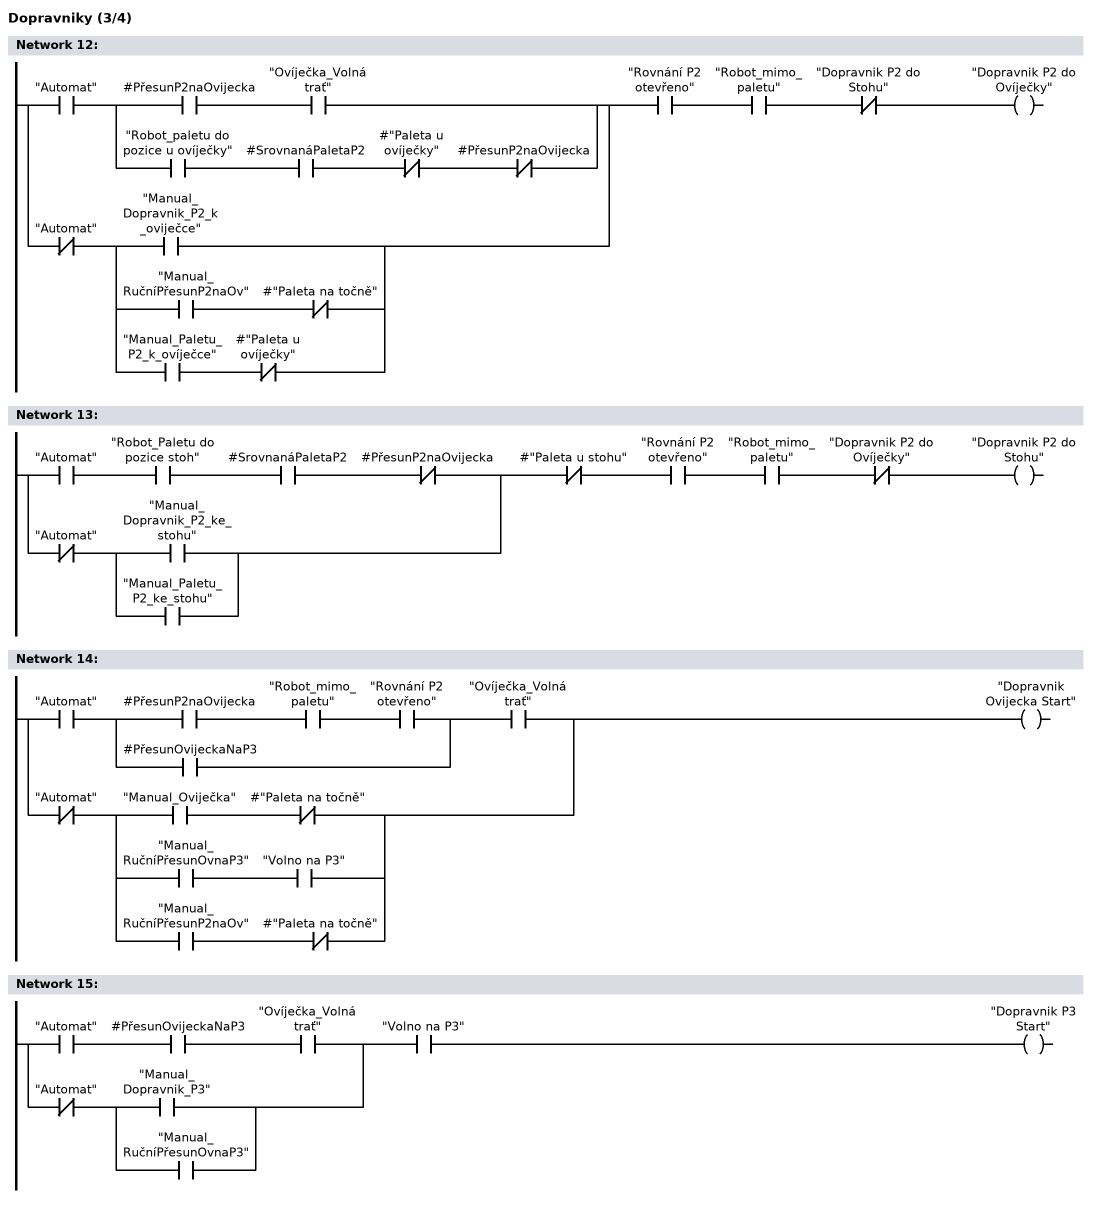
   RUNG wire#powerrail
      Contact( "Automat" )
      wire#w1
      Contact( #PřesunP2naOvijecka )
      Contact( "Ovíječka_Volná trať" )
      wire#w2
      Contact( "Rovnání P2 otevřeno" )
      Contact( "Robot_mimo_paletu" )
      I_Contact( "Dopravnik P2 do Stohu" )
      Coil( "Dopravnik P2 do Ovíječky" )
   END_RUNG
   RUNG wire#w1
      Contact( "Robot_paletu do pozice u ovíječky" )
      Contact( #SrovnanáPaletaP2 )
      I_Contact( #"Paleta u ovíječky" )
      I_Contact( #PřesunP2naOvijecka )
   END_RUNG wire#w2
   RUNG wire#powerrail
      I_Contact( "Automat" )
      wire#w3
      Contact( "Manual_Dopravnik_P2_k _oviječce" )
   END_RUNG wire#w2
   RUNG wire#w3
      Contact( "Manual_RučníPřesunP2naOv" )
      I_Contact( #"Paleta na točně" )
   END_RUNG wire#w2
   RUNG wire#w3
      Contact( "Manual_Paletu_P2_k_ovíječce" )
      I_Contact( #"Paleta u ovíječky" )
   END_RUNG wire#w2
   // the same network as SCL:
   "Dopravnik P2 do Ovíječky" := (("Automat" AND ((#PřesunP2naOvijecka AND "Ovíječka_Volná trať") OR ("Robot_paletu do pozice u ovíječky" AND #SrovnanáPaletaP2 AND NOT #"Paleta u ovíječky" AND NOT #PřesunP2naOvijecka))) OR (NOT "Automat" AND ("Manual_Dopravnik_P2_k _oviječce" OR ("Manual_RučníPřesunP2naOv" AND NOT #"Paleta na točně") OR ("Manual_Paletu_P2_k_ovíječce" AND NOT #"Paleta u ovíječky")))) AND "Rovnání P2 otevřeno" AND "Robot_mimo_paletu" AND NOT "Dopravnik P2 do Stohu";
END_REGION

REGION Network 13
   RUNG wire#powerrail
      Contact( "Automat" )
      Contact( "Robot_Paletu do pozice stoh" )
      Contact( #SrovnanáPaletaP2 )
      I_Contact( #PřesunP2naOvijecka )
      wire#w1
      I_Contact( #"Paleta u stohu" )
      Contact( "Rovnání P2 otevřeno" )
      Contact( "Robot_mimo_paletu" )
      I_Contact( "Dopravnik P2 do Ovíječky" )
      Coil( "Dopravnik P2 do Stohu" )
   END_RUNG
   RUNG wire#powerrail
      I_Contact( "Automat" )
      wire#w2
      Contact( "Manual_Dopravnik_P2_ke_stohu" )
   END_RUNG wire#w1
   RUNG wire#w2
      Contact( "Manual_Paletu_P2_ke_stohu" )
   END_RUNG wire#w1
   // the same network as SCL:
   "Dopravnik P2 do Stohu" := (("Automat" AND "Robot_Paletu do pozice stoh" AND #SrovnanáPaletaP2 AND NOT #PřesunP2naOvijecka) OR (NOT "Automat" AND ("Manual_Dopravnik_P2_ke_stohu" OR "Manual_Paletu_P2_ke_stohu"))) AND NOT #"Paleta u stohu" AND "Rovnání P2 otevřeno" AND "Robot_mimo_paletu" AND NOT "Dopravnik P2 do Ovíječky";
END_REGION

REGION Network 14
   RUNG wire#powerrail
      Contact( "Automat" )
      wire#w1
      Contact( #PřesunP2naOvijecka )
      Contact( "Robot_mimo_paletu" )
      Contact( "Rovnání P2 otevřeno" )
      wire#w2
      Contact( "Ovíječka_Volná trať" )
      wire#w3
      Coil( "Dopravnik Ovijecka Start" )
   END_RUNG
   RUNG wire#w1
      Contact( #PřesunOvijeckaNaP3 )
   END_RUNG wire#w2
   RUNG wire#powerrail
      I_Contact( "Automat" )
      wire#w4
      Contact( "Manual_Oviječka" )
      I_Contact( #"Paleta na točně" )
   END_RUNG wire#w3
   RUNG wire#w4
      Contact( "Manual_RučníPřesunOvnaP3" )
      Contact( "Volno na P3" )
   END_RUNG wire#w3
   RUNG wire#w4
      Contact( "Manual_RučníPřesunP2naOv" )
      I_Contact( #"Paleta na točně" )
   END_RUNG wire#w3
   // the same network as SCL:
   "Dopravnik Ovijecka Start" := ("Automat" AND ((#PřesunP2naOvijecka AND "Robot_mimo_paletu" AND "Rovnání P2 otevřeno") OR #PřesunOvijeckaNaP3) AND "Ovíječka_Volná trať") OR (NOT "Automat" AND (("Manual_Oviječka" AND NOT #"Paleta na točně") OR ("Manual_RučníPřesunOvnaP3" AND "Volno na P3") OR ("Manual_RučníPřesunP2naOv" AND NOT #"Paleta na točně")));
END_REGION

REGION Network 15
   RUNG wire#powerrail
      Contact( "Automat" )
      Contact( #PřesunOvijeckaNaP3 )
      Contact( "Ovíječka_Volná trať" )
      wire#w1
      Contact( "Volno na P3" )
      Coil( "Dopravnik P3 Start" )
   END_RUNG
   RUNG wire#powerrail
      I_Contact( "Automat" )
      wire#w2
      Contact( "Manual_Dopravnik_P3" )
   END_RUNG wire#w1
   RUNG wire#w2
      Contact( "Manual_RučníPřesunOvnaP3" )
   END_RUNG wire#w1
   // the same network as SCL:
   "Dopravnik P3 Start" := (("Automat" AND #PřesunOvijeckaNaP3 AND "Ovíječka_Volná trať") OR (NOT "Automat" AND ("Manual_Dopravnik_P3" OR "Manual_RučníPřesunOvnaP3"))) AND "Volno na P3";
END_REGION

REGION Network 17
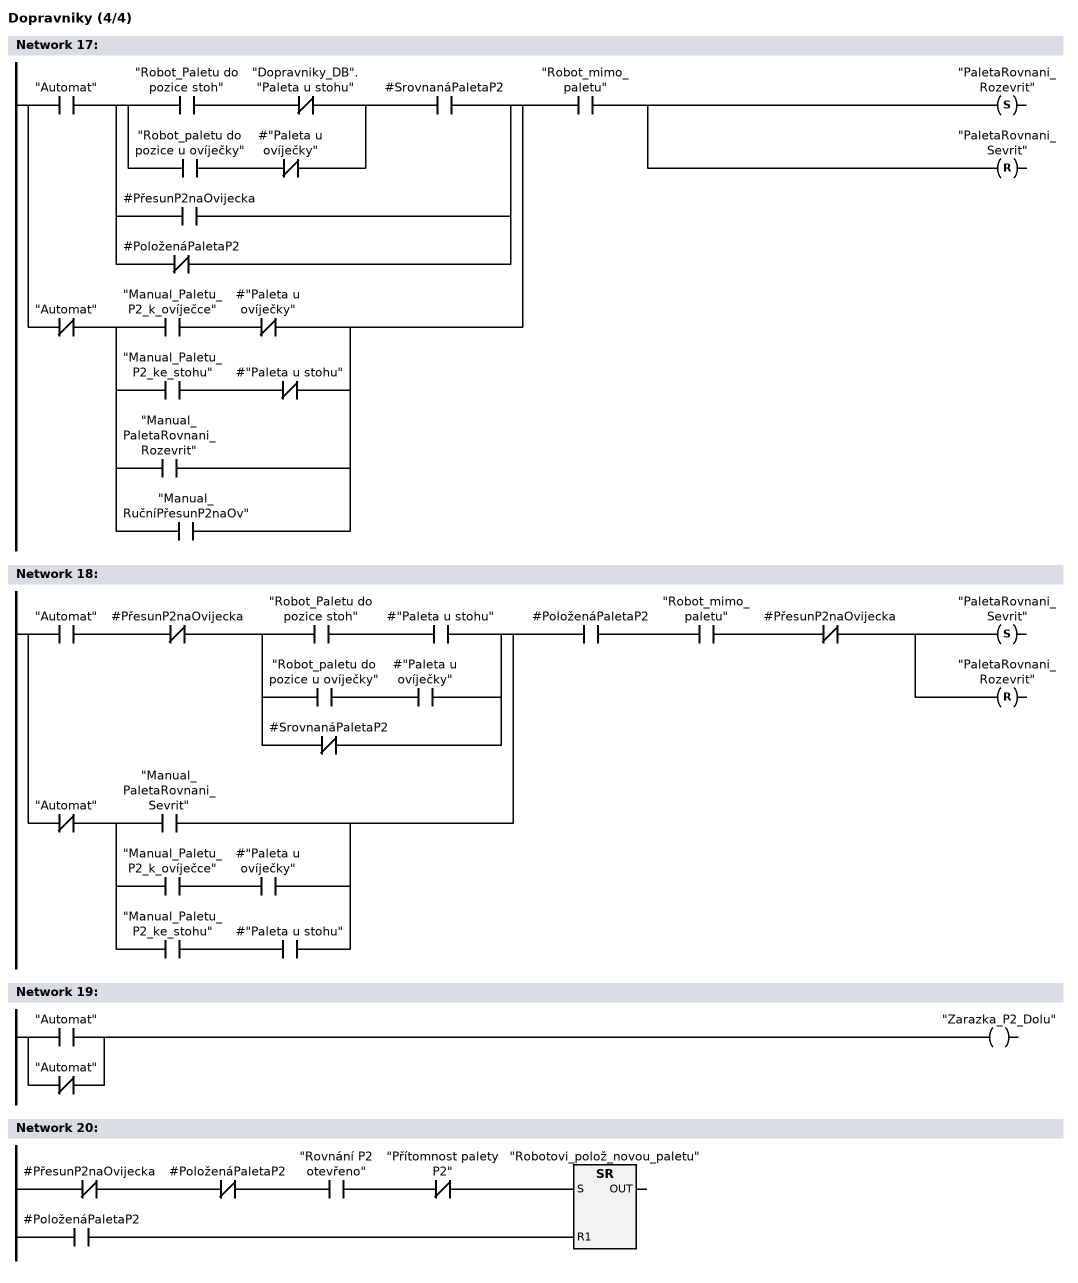
   RUNG wire#powerrail
      Contact( "Automat" )
      wire#w1
      Contact( "Robot_Paletu do pozice stoh" )
      I_Contact( "Dopravniky_DB"."Paleta u stohu" )
      wire#w2
      Contact( #SrovnanáPaletaP2 )
      wire#w3
      Contact( "Robot_mimo_paletu" )
      wire#w5
      S_Coil( "PaletaRovnani_Rozevrit" )
   END_RUNG
   RUNG wire#w1
      Contact( "Robot_paletu do pozice u ovíječky" )
      I_Contact( #"Paleta u ovíječky" )
   END_RUNG wire#w2
   RUNG wire#w1
      Contact( #PřesunP2naOvijecka )
   END_RUNG wire#w3
   RUNG wire#w1
      I_Contact( #PoloženáPaletaP2 )
   END_RUNG wire#w3
   RUNG wire#powerrail
      I_Contact( "Automat" )
      wire#w4
      Contact( "Manual_Paletu_P2_k_ovíječce" )
      I_Contact( #"Paleta u ovíječky" )
   END_RUNG wire#w3
   RUNG wire#w4
      Contact( "Manual_Paletu_P2_ke_stohu" )
      I_Contact( #"Paleta u stohu" )
   END_RUNG wire#w3
   RUNG wire#w4
      Contact( "Manual_PaletaRovnani_Rozevrit" )
   END_RUNG wire#w3
   RUNG wire#w4
      Contact( "Manual_RučníPřesunP2naOv" )
   END_RUNG wire#w3
   RUNG wire#w5
      R_Coil( "PaletaRovnani_Sevrit" )
   END_RUNG
   // the same network as SCL:
   IF (("Automat" AND (((("Robot_Paletu do pozice stoh" AND NOT "Dopravniky_DB"."Paleta u stohu") OR ("Robot_paletu do pozice u ovíječky" AND NOT #"Paleta u ovíječky")) AND #SrovnanáPaletaP2) OR #PřesunP2naOvijecka OR NOT #PoloženáPaletaP2)) OR (NOT "Automat" AND (("Manual_Paletu_P2_k_ovíječce" AND NOT #"Paleta u ovíječky") OR ("Manual_Paletu_P2_ke_stohu" AND NOT #"Paleta u stohu") OR "Manual_PaletaRovnani_Rozevrit" OR "Manual_RučníPřesunP2naOv"))) AND "Robot_mimo_paletu" THEN
       "PaletaRovnani_Rozevrit" := TRUE;
       "PaletaRovnani_Sevrit" := FALSE;
   END_IF;
END_REGION

REGION Network 18
   RUNG wire#powerrail
      Contact( "Automat" )
      I_Contact( #PřesunP2naOvijecka )
      wire#w1
      Contact( "Robot_Paletu do pozice stoh" )
      Contact( #"Paleta u stohu" )
      wire#w2
      Contact( #PoloženáPaletaP2 )
      Contact( "Robot_mimo_paletu" )
      I_Contact( #PřesunP2naOvijecka )
      wire#w4
      S_Coil( "PaletaRovnani_Sevrit" )
   END_RUNG
   RUNG wire#w1
      Contact( "Robot_paletu do pozice u ovíječky" )
      Contact( #"Paleta u ovíječky" )
   END_RUNG wire#w2
   RUNG wire#w1
      I_Contact( #SrovnanáPaletaP2 )
   END_RUNG wire#w2
   RUNG wire#powerrail
      I_Contact( "Automat" )
      wire#w3
      Contact( "Manual_PaletaRovnani_Sevrit" )
   END_RUNG wire#w2
   RUNG wire#w3
      Contact( "Manual_Paletu_P2_k_ovíječce" )
      Contact( #"Paleta u ovíječky" )
   END_RUNG wire#w2
   RUNG wire#w3
      Contact( "Manual_Paletu_P2_ke_stohu" )
      Contact( #"Paleta u stohu" )
   END_RUNG wire#w2
   RUNG wire#w4
      R_Coil( "PaletaRovnani_Rozevrit" )
   END_RUNG
   // the same network as SCL:
   IF (("Automat" AND NOT #PřesunP2naOvijecka AND (("Robot_Paletu do pozice stoh" AND #"Paleta u stohu") OR ("Robot_paletu do pozice u ovíječky" AND #"Paleta u ovíječky") OR NOT #SrovnanáPaletaP2)) OR (NOT "Automat" AND ("Manual_PaletaRovnani_Sevrit" OR ("Manual_Paletu_P2_k_ovíječce" AND #"Paleta u ovíječky") OR ("Manual_Paletu_P2_ke_stohu" AND #"Paleta u stohu")))) AND #PoloženáPaletaP2 AND "Robot_mimo_paletu" AND NOT #PřesunP2naOvijecka THEN
       "PaletaRovnani_Sevrit" := TRUE;
       "PaletaRovnani_Rozevrit" := FALSE;
   END_IF;
END_REGION

REGION Network 19
   RUNG wire#powerrail
      Contact( "Automat" )
      wire#w1
      Coil( "Zarazka_P2_Dolu" )
   END_RUNG
   RUNG wire#powerrail
      I_Contact( "Automat" )
   END_RUNG wire#w1
   // the same network as SCL:
   "Zarazka_P2_Dolu" := "Automat" OR NOT "Automat";
END_REGION

REGION Network 20
   RUNG wire#powerrail
      I_Contact( #PřesunP2naOvijecka )
      I_Contact( #PoloženáPaletaP2 )
      Contact( "Rovnání P2 otevřeno" )
      I_Contact( "Přítomnost palety P2" )
      S_SR(operand := "Robotovi_polož_novou_paletu", r1 := wire#w1)
   END_RUNG
   RUNG wire#powerrail
      Contact( #PoloženáPaletaP2 )
   END_RUNG wire#w1
   // the same network as SCL:
   IF NOT #PřesunP2naOvijecka AND NOT #PoloženáPaletaP2 AND "Rovnání P2 otevřeno" AND NOT "Přítomnost palety P2" THEN
       "Robotovi_polož_novou_paletu" := TRUE;   // SR flip-flop
   END_IF;
   IF #PoloženáPaletaP2 THEN "Robotovi_polož_novou_paletu" := FALSE; END_IF;
END_REGION
END_FUNCTION_BLOCK

FUNCTION_BLOCK "Klapky"   // FB11, LAD
TITLE = Klapky
{ S7_Optimized_Access := 'FALSE' }
VERSION : 0.1
BEGIN
END_FUNCTION_BLOCK

FUNCTION_BLOCK "Dopravníky pytlů"   // FB12, LAD
{ S7_Optimized_Access := 'FALSE' }
VERSION : 0.1
   VAR
      "Pytel na váze" : Bool;
      "Pytel na P1" : Bool;
      "Paměť 1" : Bool;
      "Paměť 2" : Bool;
      "Paměť 3" : Bool;
      "Paměť 4" : Bool;
      "Time" : S5Time := S5T#400ms;
      "Vadný pytel na váze" : Bool;
      "Vadný pytel na P1" : Bool;
      "Dopravník váha start" : Bool;
      "Dopravnik váha stop" : Bool;
   END_VAR
   VAR_TEMP   // added for the SCL form of the ladder/FBD networks
      _w1 : Bool;
      _s5time1 : S5Time;
      _w2 : Bool;
      _s5time2 : S5Time;
      _w3 : Bool;
      _w4 : Bool;
      _w5 : Bool;
      _s5time3 : S5Time;
   END_VAR
BEGIN

REGION Network 1
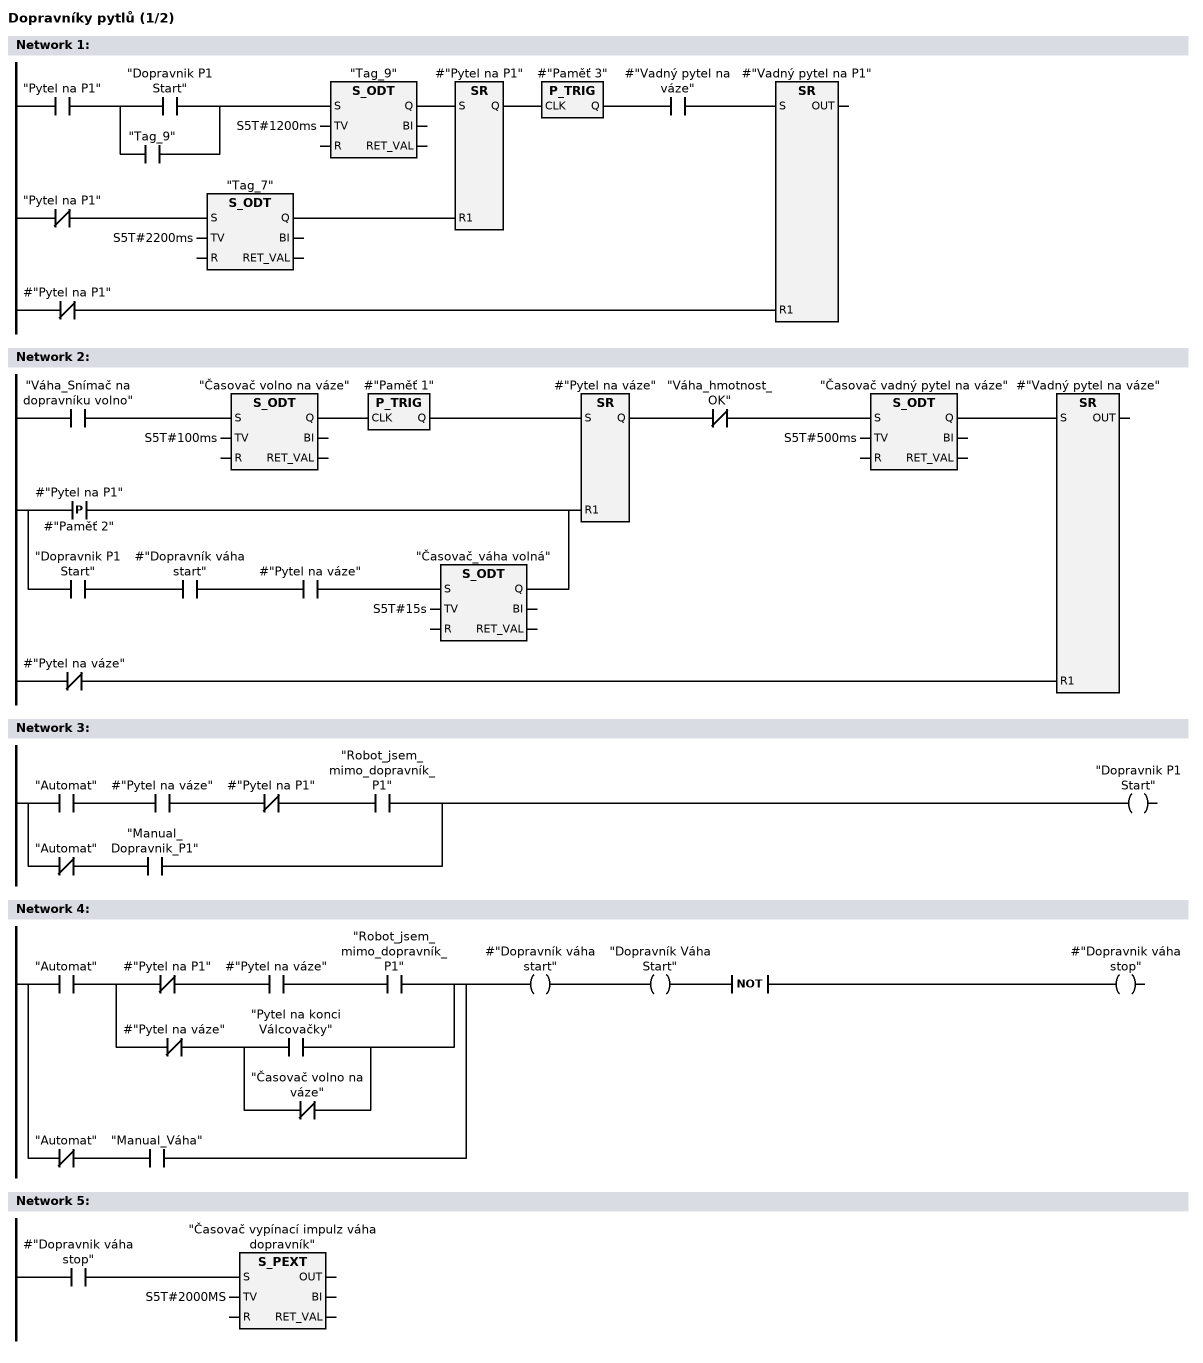
   RUNG wire#powerrail
      Contact( "Pytel na P1" )
      wire#w1
      Contact( "Dopravnik P1 Start" )
      wire#w2
      S_ODT(T_NO := "Tag_9", TV := S5T#1200ms, R :=, BI =>, RET_VAL =>)
      S_SR(operand := #"Pytel na P1", r1 := wire#w3)
      P_Trig( #"Paměť 3" )
      Contact( #"Vadný pytel na váze" )
      S_SR(operand := #"Vadný pytel na P1", r1 := wire#w4)
   END_RUNG
   RUNG wire#w1
      Contact( "Tag_9" )
   END_RUNG wire#w2
   RUNG wire#powerrail
      I_Contact( "Pytel na P1" )
      S_ODT(T_NO := "Tag_7", TV := S5T#2200ms, R :=, BI =>, RET_VAL =>)
   END_RUNG wire#w3
   RUNG wire#powerrail
      I_Contact( #"Pytel na P1" )
   END_RUNG wire#w4
   // the same network as SCL:
   #_s5time1 := S_ODT(T_NO := "Tag_9",
                      S := "Pytel na P1" AND ("Dopravnik P1 Start" OR "Tag_9"),
                      TV := S5T#1200ms,
                      Q => #_w1);
   #_s5time2 := S_ODT(T_NO := "Tag_7", S := NOT "Pytel na P1", TV := S5T#2200ms, Q => #_w2);
   IF #_w1 THEN
       #"Pytel na P1" := TRUE;   // SR flip-flop
   END_IF;
   IF #_w2 THEN #"Pytel na P1" := FALSE; END_IF;
   #_w3 := #"Pytel na P1" AND NOT #"Paměť 3";   // rising edge
   #"Paměť 3" := #"Pytel na P1";
   IF #_w3 AND #"Vadný pytel na váze" THEN
       #"Vadný pytel na P1" := TRUE;   // SR flip-flop
   END_IF;
   IF NOT #"Pytel na P1" THEN #"Vadný pytel na P1" := FALSE; END_IF;
END_REGION

REGION Network 2
   RUNG wire#powerrail
      Contact( "Váha_Snímač na dopravníku volno" )
      S_ODT(T_NO := "Časovač volno na váze", TV := S5T#100ms, R :=, BI =>, RET_VAL =>)
      P_Trig( #"Paměť 1" )
      S_SR(operand := #"Pytel na váze", r1 := wire#w1)
      I_Contact( "Váha_hmotnost_OK" )
      S_ODT(T_NO := "Časovač vadný pytel na váze", TV := S5T#500ms, R :=, BI =>, RET_VAL =>)
      S_SR(operand := #"Vadný pytel na váze", r1 := wire#w2)
   END_RUNG
   RUNG wire#powerrail
      P_Contact(operand := #"Pytel na P1", bit := #"Paměť 2")
   END_RUNG wire#w1
   RUNG wire#powerrail
      Contact( "Dopravnik P1 Start" )
      Contact( #"Dopravník váha start" )
      Contact( #"Pytel na váze" )
      S_ODT(T_NO := "Časovač_váha volná", TV := S5T#15s, R :=, BI =>, RET_VAL =>)
   END_RUNG wire#w1
   RUNG wire#powerrail
      I_Contact( #"Pytel na váze" )
   END_RUNG wire#w2
   // the same network as SCL:
   #_s5time1 := S_ODT(T_NO := "Časovač volno na váze",
                      S := "Váha_Snímač na dopravníku volno",
                      TV := S5T#100ms,
                      Q => #_w1);
   #_w2 := #_w1 AND NOT #"Paměť 1";   // rising edge
   #"Paměť 1" := #_w1;
   #_w3 := #"Pytel na P1" AND NOT #"Paměť 2";   // rising edge of #"Pytel na P1"
   #"Paměť 2" := #"Pytel na P1";
   #_s5time2 := S_ODT(T_NO := "Časovač_váha volná",
                      S := "Dopravnik P1 Start" AND #"Dopravník váha start" AND #"Pytel na váze",
                      TV := S5T#15s,
                      Q => #_w4);
   IF #_w2 THEN
       #"Pytel na váze" := TRUE;   // SR flip-flop
   END_IF;
   IF #_w3 OR #_w4 THEN #"Pytel na váze" := FALSE; END_IF;
   #_s5time3 := S_ODT(T_NO := "Časovač vadný pytel na váze",
                      S := #"Pytel na váze" AND NOT "Váha_hmotnost_OK",
                      TV := S5T#500ms,
                      Q => #_w5);
   IF #_w5 THEN
       #"Vadný pytel na váze" := TRUE;   // SR flip-flop
   END_IF;
   IF NOT #"Pytel na váze" THEN #"Vadný pytel na váze" := FALSE; END_IF;
END_REGION

REGION Network 3
   RUNG wire#powerrail
      Contact( "Automat" )
      Contact( #"Pytel na váze" )
      I_Contact( #"Pytel na P1" )
      Contact( "Robot_jsem_mimo_dopravník_P1" )
      wire#w1
      Coil( "Dopravnik P1 Start" )
   END_RUNG
   RUNG wire#powerrail
      I_Contact( "Automat" )
      Contact( "Manual_Dopravnik_P1" )
   END_RUNG wire#w1
   // the same network as SCL:
   "Dopravnik P1 Start" := ("Automat" AND #"Pytel na váze" AND NOT #"Pytel na P1" AND "Robot_jsem_mimo_dopravník_P1") OR (NOT "Automat" AND "Manual_Dopravnik_P1");
END_REGION

REGION Network 4
   RUNG wire#powerrail
      Contact( "Automat" )
      wire#w1
      I_Contact( #"Pytel na P1" )
      Contact( #"Pytel na váze" )
      Contact( "Robot_jsem_mimo_dopravník_P1" )
      wire#w2
      Coil( #"Dopravník váha start" )
      Coil( "Dopravník Váha Start" )
      Not()
      Coil( #"Dopravnik váha stop" )
   END_RUNG
   RUNG wire#w1
      I_Contact( #"Pytel na váze" )
      wire#w3
      Contact( "Pytel na konci Válcovačky" )
   END_RUNG wire#w2
   RUNG wire#w3
      I_Contact( "Časovač volno na váze" )
   END_RUNG wire#w2
   RUNG wire#powerrail
      I_Contact( "Automat" )
      Contact( "Manual_Váha" )
   END_RUNG wire#w2
   // the same network as SCL:
   #"Dopravník váha start" := ("Automat" AND ((NOT #"Pytel na P1" AND #"Pytel na váze" AND "Robot_jsem_mimo_dopravník_P1") OR (NOT #"Pytel na váze" AND ("Pytel na konci Válcovačky" OR NOT "Časovač volno na váze")))) OR (NOT "Automat" AND "Manual_Váha");
   "Dopravník Váha Start" := #"Dopravník váha start";
   #"Dopravnik váha stop" := NOT #"Dopravník váha start";
END_REGION

REGION Network 5
   RUNG wire#powerrail
      Contact( #"Dopravnik váha stop" )
      S_PEXT(T_NO := "Časovač vypínací impulz váha dopravník", TV := S5T#2000MS, R :=, BI =>, RET_VAL =>)
   END_RUNG
   // the same network as SCL:
   #_s5time1 := S_PEXT(T_NO := "Časovač vypínací impulz váha dopravník",
                       S := #"Dopravnik váha stop",
                       TV := S5T#2000MS);
END_REGION

REGION Network 6
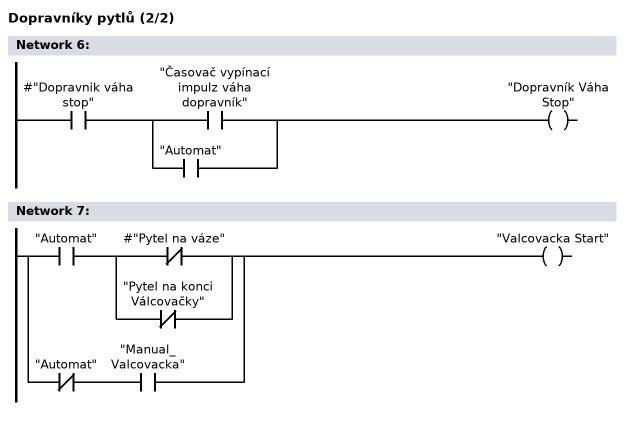
   RUNG wire#powerrail
      Contact( #"Dopravnik váha stop" )
      wire#w1
      Contact( "Časovač vypínací impulz váha dopravník" )
      wire#w2
      Coil( "Dopravník Váha Stop" )
   END_RUNG
   RUNG wire#w1
      Contact( "Automat" )
   END_RUNG wire#w2
   // the same network as SCL:
   "Dopravník Váha Stop" := #"Dopravnik váha stop" AND ("Časovač vypínací impulz váha dopravník" OR "Automat");
END_REGION

REGION Network 7
   RUNG wire#powerrail
      Contact( "Automat" )
      wire#w1
      I_Contact( #"Pytel na váze" )
      wire#w2
      Coil( "Valcovacka Start" )
   END_RUNG
   RUNG wire#w1
      I_Contact( "Pytel na konci Válcovačky" )
   END_RUNG wire#w2
   RUNG wire#powerrail
      I_Contact( "Automat" )
      Contact( "Manual_Valcovacka" )
   END_RUNG wire#w2
   // the same network as SCL:
   "Valcovacka Start" := ("Automat" AND (NOT #"Pytel na váze" OR NOT "Pytel na konci Válcovačky")) OR (NOT "Automat" AND "Manual_Valcovacka");
END_REGION
END_FUNCTION_BLOCK

FUNCTION_BLOCK "Komunikace ovijecka"   // FB50, LAD
{ S7_Optimized_Access := 'FALSE' }
VERSION : 0.1
BEGIN
END_FUNCTION_BLOCK

FUNCTION_BLOCK "Komunikace robot"   // FB51, LAD
{ S7_Optimized_Access := 'FALSE' }
VERSION : 0.1
   VAR
      Položená_paleta_na_P2 : Bool;
      Plná_paleta_P2 : Bool;
      "PHrana_plná paleta" : Bool;
      "Paměť hrana paleta vadných plná" : Bool;
      "Paměť hrana prázdný stohovač palet" : Bool;
   END_VAR
   VAR_TEMP
      Robot_paleta_uložena : Bool;
      Robot_plná_paleta : Bool;
      Temp_1 : Byte;
      Temp_2 : Array[0..5] of Byte;
      index : Byte;
   END_VAR
   VAR_TEMP   // added for the SCL form of the ladder/FBD networks
      _w1 : Bool;
      _s5time1 : S5Time;
      _w2 : Bool;
      _s5time2 : S5Time;
   END_VAR
BEGIN

REGION Network 1
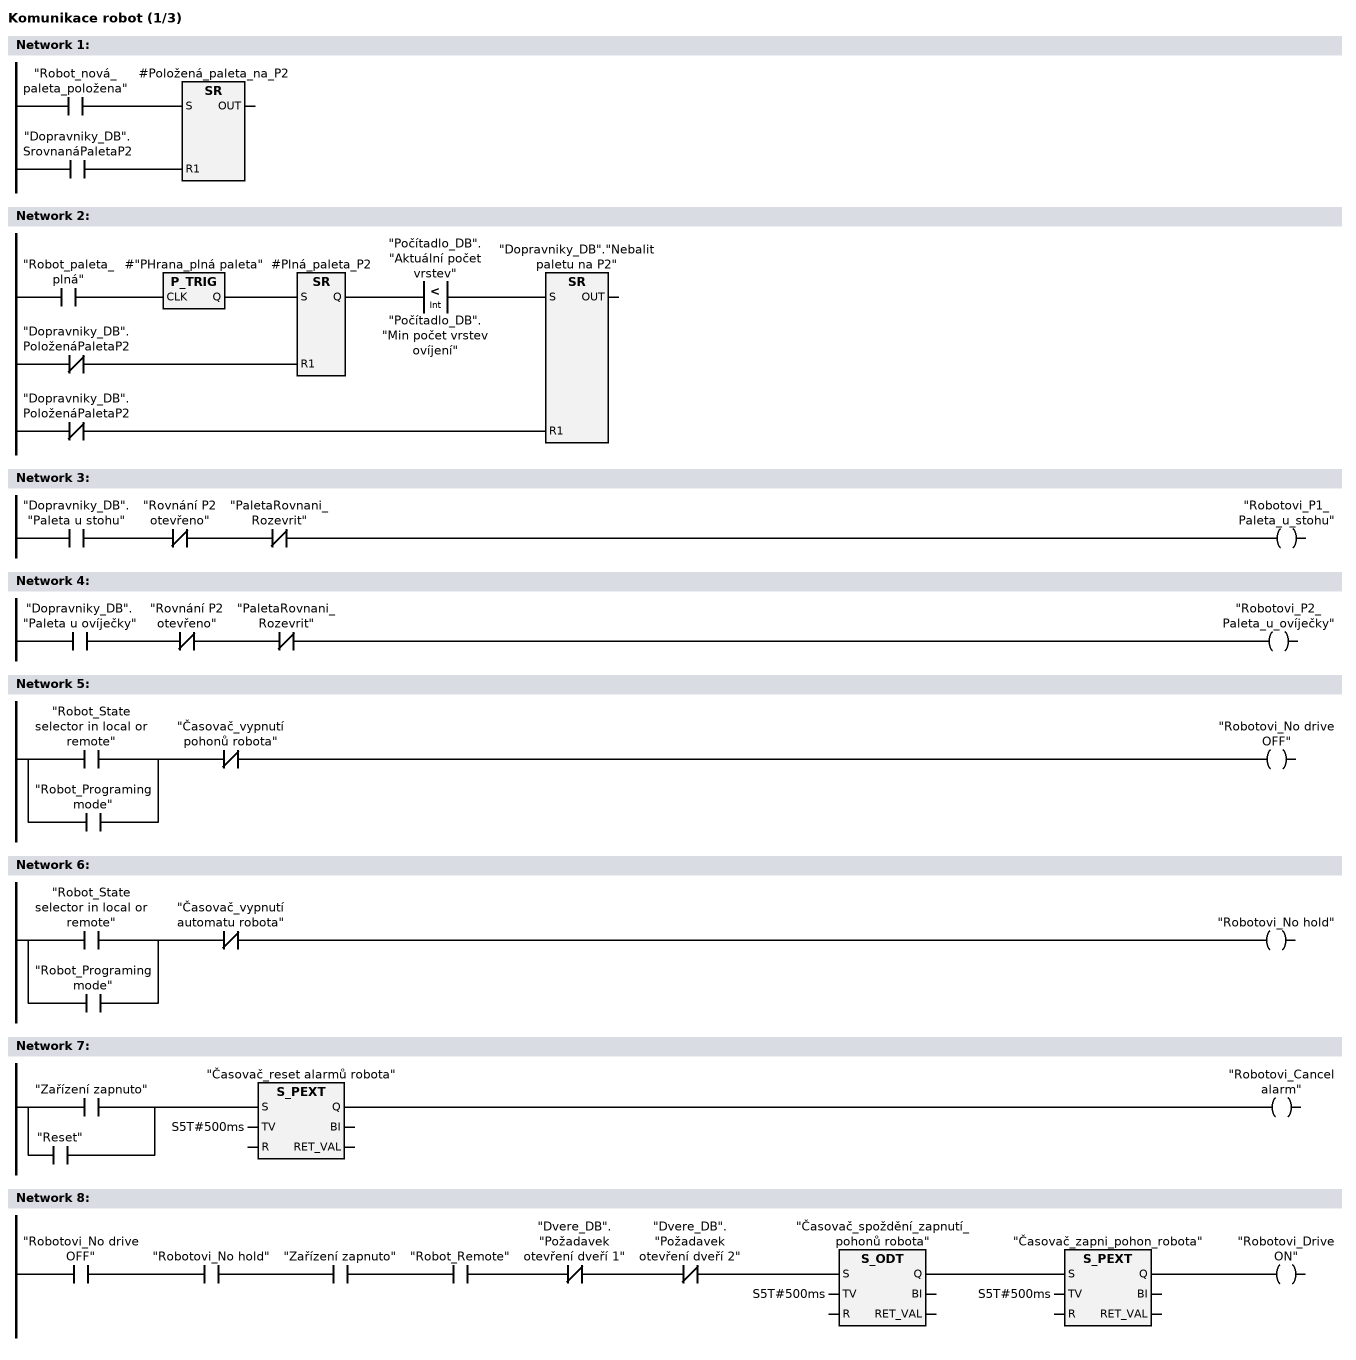
   RUNG wire#powerrail
      Contact( "Robot_nová_paleta_položena" )
      S_SR(operand := #Položená_paleta_na_P2, r1 := wire#w1)
   END_RUNG
   RUNG wire#powerrail
      Contact( "Dopravniky_DB".SrovnanáPaletaP2 )
   END_RUNG wire#w1
   // the same network as SCL:
   IF "Robot_nová_paleta_položena" THEN
       #Položená_paleta_na_P2 := TRUE;   // SR flip-flop
   END_IF;
   IF "Dopravniky_DB".SrovnanáPaletaP2 THEN #Položená_paleta_na_P2 := FALSE; END_IF;
END_REGION

REGION Network 2
   RUNG wire#powerrail
      Contact( "Robot_paleta_plná" )
      P_Trig( #"PHrana_plná paleta" )
      S_SR(operand := #Plná_paleta_P2, r1 := wire#w1)
      { S7_Templates := "SrcType := Int" } LT_Contact(in1 := "Počítadlo_DB"."Aktuální počet vrstev", in2 := "Počítadlo_DB"."Min počet vrstev ovíjení")
      S_SR(operand := "Dopravniky_DB"."Nebalit paletu na P2", r1 := wire#w2)
   END_RUNG
   RUNG wire#powerrail
      I_Contact( "Dopravniky_DB".PoloženáPaletaP2 )
   END_RUNG wire#w1
   RUNG wire#powerrail
      I_Contact( "Dopravniky_DB".PoloženáPaletaP2 )
   END_RUNG wire#w2
   // the same network as SCL:
   #_w1 := "Robot_paleta_plná" AND NOT #"PHrana_plná paleta";   // rising edge
   #"PHrana_plná paleta" := "Robot_paleta_plná";
   IF #_w1 THEN
       #Plná_paleta_P2 := TRUE;   // SR flip-flop
   END_IF;
   IF NOT "Dopravniky_DB".PoloženáPaletaP2 THEN #Plná_paleta_P2 := FALSE; END_IF;
   IF #Plná_paleta_P2 AND ("Počítadlo_DB"."Aktuální počet vrstev" < "Počítadlo_DB"."Min počet vrstev ovíjení") THEN
       "Dopravniky_DB"."Nebalit paletu na P2" := TRUE;   // SR flip-flop
   END_IF;
   IF NOT "Dopravniky_DB".PoloženáPaletaP2 THEN "Dopravniky_DB"."Nebalit paletu na P2" := FALSE; END_IF;
END_REGION

REGION Network 3
   RUNG wire#powerrail
      Contact( "Dopravniky_DB"."Paleta u stohu" )
      I_Contact( "Rovnání P2 otevřeno" )
      I_Contact( "PaletaRovnani_Rozevrit" )
      Coil( "Robotovi_P1_Paleta_u_stohu" )
   END_RUNG
   // the same network as SCL:
   "Robotovi_P1_Paleta_u_stohu" := "Dopravniky_DB"."Paleta u stohu" AND NOT "Rovnání P2 otevřeno" AND NOT "PaletaRovnani_Rozevrit";
END_REGION

REGION Network 4
   RUNG wire#powerrail
      Contact( "Dopravniky_DB"."Paleta u ovíječky" )
      I_Contact( "Rovnání P2 otevřeno" )
      I_Contact( "PaletaRovnani_Rozevrit" )
      Coil( "Robotovi_P2_Paleta_u_ovíječky" )
   END_RUNG
   // the same network as SCL:
   "Robotovi_P2_Paleta_u_ovíječky" := "Dopravniky_DB"."Paleta u ovíječky" AND NOT "Rovnání P2 otevřeno" AND NOT "PaletaRovnani_Rozevrit";
END_REGION

REGION Network 5
   RUNG wire#powerrail
      Contact( "Robot_State selector in local or remote" )
      wire#w1
      I_Contact( "Časovač_vypnutí pohonů robota" )
      Coil( "Robotovi_No drive OFF" )
   END_RUNG
   RUNG wire#powerrail
      Contact( "Robot_Programing mode" )
   END_RUNG wire#w1
   // the same network as SCL:
   "Robotovi_No drive OFF" := ("Robot_State selector in local or remote" OR "Robot_Programing mode") AND NOT "Časovač_vypnutí pohonů robota";
END_REGION

REGION Network 6
   RUNG wire#powerrail
      Contact( "Robot_State selector in local or remote" )
      wire#w1
      I_Contact( "Časovač_vypnutí automatu robota" )
      Coil( "Robotovi_No hold" )
   END_RUNG
   RUNG wire#powerrail
      Contact( "Robot_Programing mode" )
   END_RUNG wire#w1
   // the same network as SCL:
   "Robotovi_No hold" := ("Robot_State selector in local or remote" OR "Robot_Programing mode") AND NOT "Časovač_vypnutí automatu robota";
END_REGION

REGION Network 7
   RUNG wire#powerrail
      Contact( "Zařízení zapnuto" )
      wire#w1
      S_PEXT(T_NO := "Časovač_reset alarmů robota", TV := S5T#500ms, R :=, BI =>, RET_VAL =>)
      Coil( "Robotovi_Cancel alarm" )
   END_RUNG
   RUNG wire#powerrail
      Contact( "Reset" )
   END_RUNG wire#w1
   // the same network as SCL:
   #_s5time1 := S_PEXT(T_NO := "Časovač_reset alarmů robota",
                       S := "Zařízení zapnuto" OR "Reset",
                       TV := S5T#500ms,
                       Q => #_w1);
   "Robotovi_Cancel alarm" := #_w1;
END_REGION

REGION Network 8
   RUNG wire#powerrail
      Contact( "Robotovi_No drive OFF" )
      Contact( "Robotovi_No hold" )
      Contact( "Zařízení zapnuto" )
      Contact( "Robot_Remote" )
      I_Contact( "Dvere_DB"."Požadavek otevření dveří 1" )
      I_Contact( "Dvere_DB"."Požadavek otevření dveří 2" )
      S_ODT(T_NO := "Časovač_spoždění_zapnutí_pohonů robota", TV := S5T#500ms, R :=, BI =>, RET_VAL =>)
      S_PEXT(T_NO := "Časovač_zapni_pohon_robota", TV := S5T#500ms, R :=, BI =>, RET_VAL =>)
      Coil( "Robotovi_Drive ON" )
   END_RUNG
   // the same network as SCL:
   #_s5time1 := S_ODT(T_NO := "Časovač_spoždění_zapnutí_pohonů robota",
                      S := "Robotovi_No drive OFF" AND "Robotovi_No hold" AND "Zařízení zapnuto" AND "Robot_Remote" AND NOT "Dvere_DB"."Požadavek otevření dveří 1" AND NOT "Dvere_DB"."Požadavek otevření dveří 2",
                      TV := S5T#500ms,
                      Q => #_w1);
   #_s5time2 := S_PEXT(T_NO := "Časovač_zapni_pohon_robota", S := #_w1, TV := S5T#500ms, Q => #_w2);
   "Robotovi_Drive ON" := #_w2;
END_REGION

REGION Network 9
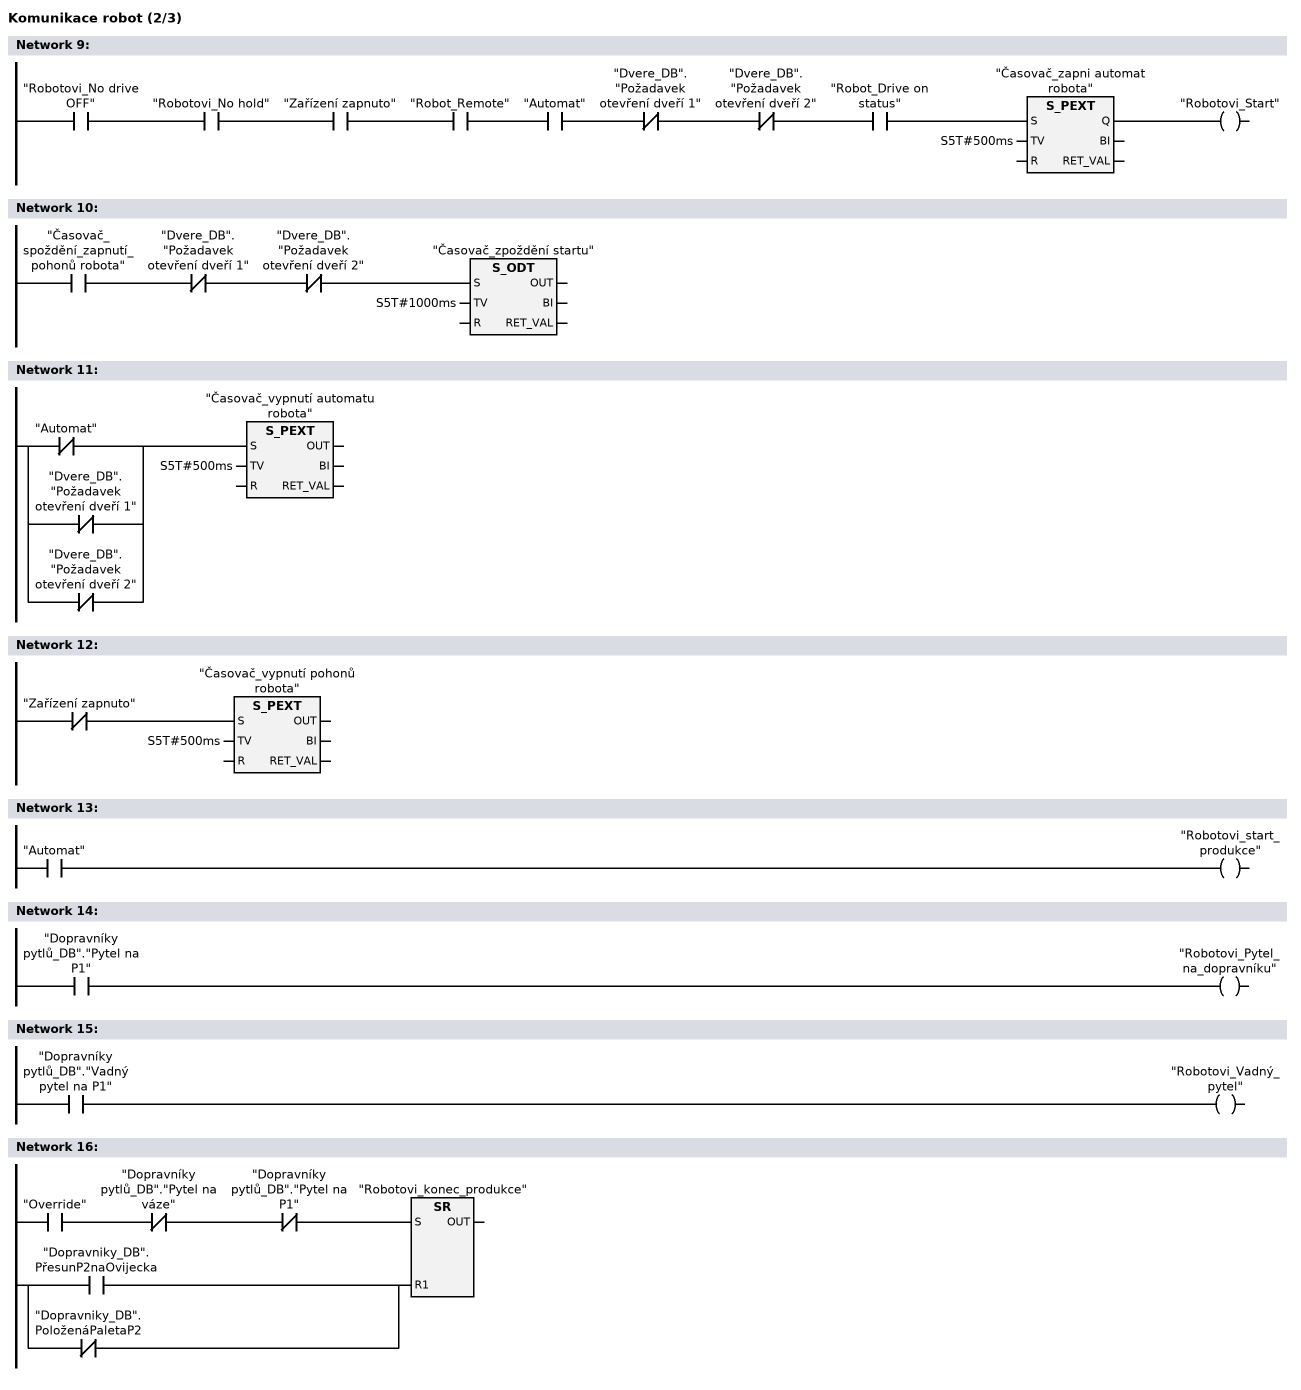
   RUNG wire#powerrail
      Contact( "Robotovi_No drive OFF" )
      Contact( "Robotovi_No hold" )
      Contact( "Zařízení zapnuto" )
      Contact( "Robot_Remote" )
      Contact( "Automat" )
      I_Contact( "Dvere_DB"."Požadavek otevření dveří 1" )
      I_Contact( "Dvere_DB"."Požadavek otevření dveří 2" )
      Contact( "Robot_Drive on status" )
      S_PEXT(T_NO := "Časovač_zapni automat robota", TV := S5T#500ms, R :=, BI =>, RET_VAL =>)
      Coil( "Robotovi_Start" )
   END_RUNG
   // the same network as SCL:
   #_s5time1 := S_PEXT(T_NO := "Časovač_zapni automat robota",
                       S := "Robotovi_No drive OFF" AND "Robotovi_No hold" AND "Zařízení zapnuto" AND "Robot_Remote" AND "Automat" AND NOT "Dvere_DB"."Požadavek otevření dveří 1" AND NOT "Dvere_DB"."Požadavek otevření dveří 2" AND "Robot_Drive on status",
                       TV := S5T#500ms,
                       Q => #_w1);
   "Robotovi_Start" := #_w1;
END_REGION

REGION Network 10
   RUNG wire#powerrail
      Contact( "Časovač_spoždění_zapnutí_pohonů robota" )
      I_Contact( "Dvere_DB"."Požadavek otevření dveří 1" )
      I_Contact( "Dvere_DB"."Požadavek otevření dveří 2" )
      S_ODT(T_NO := "Časovač_zpoždění startu", TV := S5T#1000ms, R :=, BI =>, RET_VAL =>)
   END_RUNG
   // the same network as SCL:
   #_s5time1 := S_ODT(T_NO := "Časovač_zpoždění startu",
                      S := "Časovač_spoždění_zapnutí_pohonů robota" AND NOT "Dvere_DB"."Požadavek otevření dveří 1" AND NOT "Dvere_DB"."Požadavek otevření dveří 2",
                      TV := S5T#1000ms);
END_REGION

REGION Network 11
   RUNG wire#powerrail
      I_Contact( "Automat" )
      wire#w1
      S_PEXT(T_NO := "Časovač_vypnutí automatu robota", TV := S5T#500ms, R :=, BI =>, RET_VAL =>)
   END_RUNG
   RUNG wire#powerrail
      I_Contact( "Dvere_DB"."Požadavek otevření dveří 1" )
   END_RUNG wire#w1
   RUNG wire#powerrail
      I_Contact( "Dvere_DB"."Požadavek otevření dveří 2" )
   END_RUNG wire#w1
   // the same network as SCL:
   #_s5time1 := S_PEXT(T_NO := "Časovač_vypnutí automatu robota",
                       S := NOT "Automat" OR NOT "Dvere_DB"."Požadavek otevření dveří 1" OR NOT "Dvere_DB"."Požadavek otevření dveří 2",
                       TV := S5T#500ms);
END_REGION

REGION Network 12
   RUNG wire#powerrail
      I_Contact( "Zařízení zapnuto" )
      S_PEXT(T_NO := "Časovač_vypnutí pohonů robota", TV := S5T#500ms, R :=, BI =>, RET_VAL =>)
   END_RUNG
   // the same network as SCL:
   #_s5time1 := S_PEXT(T_NO := "Časovač_vypnutí pohonů robota", S := NOT "Zařízení zapnuto", TV := S5T#500ms);
END_REGION

REGION Network 13
   RUNG wire#powerrail
      Contact( "Automat" )
      Coil( "Robotovi_start_produkce" )
   END_RUNG
   // the same network as SCL:
   "Robotovi_start_produkce" := "Automat";
END_REGION

REGION Network 14
   RUNG wire#powerrail
      Contact( "Dopravníky pytlů_DB"."Pytel na P1" )
      Coil( "Robotovi_Pytel_na_dopravníku" )
   END_RUNG
   // the same network as SCL:
   "Robotovi_Pytel_na_dopravníku" := "Dopravníky pytlů_DB"."Pytel na P1";
END_REGION

REGION Network 15
   RUNG wire#powerrail
      Contact( "Dopravníky pytlů_DB"."Vadný pytel na P1" )
      Coil( "Robotovi_Vadný_pytel" )
   END_RUNG
   // the same network as SCL:
   "Robotovi_Vadný_pytel" := "Dopravníky pytlů_DB"."Vadný pytel na P1";
END_REGION

REGION Network 16
   RUNG wire#powerrail
      Contact( "Override" )
      I_Contact( "Dopravníky pytlů_DB"."Pytel na váze" )
      I_Contact( "Dopravníky pytlů_DB"."Pytel na P1" )
      S_SR(operand := "Robotovi_konec_produkce", r1 := wire#w1)
   END_RUNG
   RUNG wire#powerrail
      Contact( "Dopravniky_DB".PřesunP2naOvijecka )
   END_RUNG wire#w1
   RUNG wire#powerrail
      I_Contact( "Dopravniky_DB".PoloženáPaletaP2 )
   END_RUNG wire#w1
   // the same network as SCL:
   IF "Override" AND NOT "Dopravníky pytlů_DB"."Pytel na váze" AND NOT "Dopravníky pytlů_DB"."Pytel na P1" THEN
       "Robotovi_konec_produkce" := TRUE;   // SR flip-flop
   END_IF;
   IF "Dopravniky_DB".PřesunP2naOvijecka OR NOT "Dopravniky_DB".PoloženáPaletaP2 THEN
       "Robotovi_konec_produkce" := FALSE;
   END_IF;
END_REGION

REGION Network 18
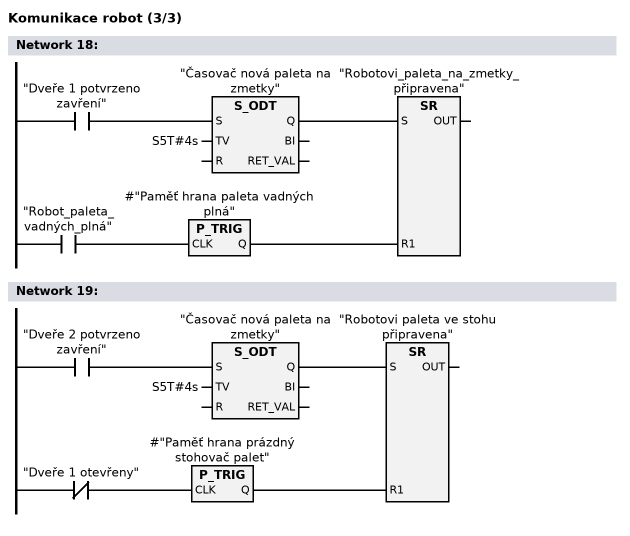
   RUNG wire#powerrail
      Contact( "Dveře 1 potvrzeno zavření" )
      S_ODT(T_NO := "Časovač nová paleta na zmetky", TV := S5T#4s, R :=, BI =>, RET_VAL =>)
      S_SR(operand := "Robotovi_paleta_na_zmetky_připravena", r1 := wire#w1)
   END_RUNG
   RUNG wire#powerrail
      Contact( "Robot_paleta_vadných_plná" )
      P_Trig( #"Paměť hrana paleta vadných plná" )
   END_RUNG wire#w1
   // the same network as SCL:
   #_s5time1 := S_ODT(T_NO := "Časovač nová paleta na zmetky",
                      S := "Dveře 1 potvrzeno zavření",
                      TV := S5T#4s,
                      Q => #_w1);
   #_w2 := "Robot_paleta_vadných_plná" AND NOT #"Paměť hrana paleta vadných plná";   // rising edge
   #"Paměť hrana paleta vadných plná" := "Robot_paleta_vadných_plná";
   IF #_w1 THEN
       "Robotovi_paleta_na_zmetky_připravena" := TRUE;   // SR flip-flop
   END_IF;
   IF #_w2 THEN "Robotovi_paleta_na_zmetky_připravena" := FALSE; END_IF;
END_REGION

REGION Network 19
   RUNG wire#powerrail
      Contact( "Dveře 2 potvrzeno zavření" )
      S_ODT(T_NO := "Časovač nová paleta na zmetky", TV := S5T#4s, R :=, BI =>, RET_VAL =>)
      S_SR(operand := "Robotovi paleta ve stohu připravena", r1 := wire#w1)
   END_RUNG
   RUNG wire#powerrail
      I_Contact( "Dveře 1 otevřeny" )
      P_Trig( #"Paměť hrana prázdný stohovač palet" )
   END_RUNG wire#w1
   // the same network as SCL:
   #_s5time1 := S_ODT(T_NO := "Časovač nová paleta na zmetky",
                      S := "Dveře 2 potvrzeno zavření",
                      TV := S5T#4s,
                      Q => #_w1);
   #_w2 := NOT "Dveře 1 otevřeny" AND NOT #"Paměť hrana prázdný stohovač palet";   // rising edge
   #"Paměť hrana prázdný stohovač palet" := NOT "Dveře 1 otevřeny";
   IF #_w1 THEN
       "Robotovi paleta ve stohu připravena" := TRUE;   // SR flip-flop
   END_IF;
   IF #_w2 THEN "Robotovi paleta ve stohu připravena" := FALSE; END_IF;
END_REGION
END_FUNCTION_BLOCK

FUNCTION_BLOCK "Komunikace vaha"   // FB53, LAD
{ S7_Optimized_Access := 'FALSE' }
VERSION : 0.1
BEGIN
END_FUNCTION_BLOCK

FUNCTION_BLOCK "Opticka zavora"   // FB54, LAD
{ S7_Optimized_Access := 'FALSE' }
VERSION : 0.1
BEGIN
END_FUNCTION_BLOCK

FUNCTION_BLOCK "Dvere"   // FB60, LAD
{ S7_Optimized_Access := 'FALSE' }
VERSION : 0.1
   VAR
      "Požadavek otevření dveří 1" : Bool;
      "Požadavek otevření dveří 2" : Bool;
   END_VAR
BEGIN

REGION Network 1
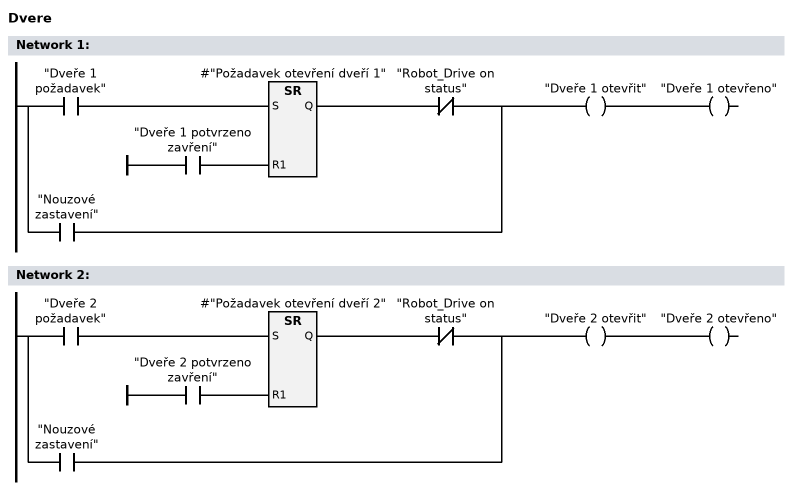
   RUNG wire#powerrail
      Contact( "Dveře 1 požadavek" )
      S_SR(operand := #"Požadavek otevření dveří 1", r1 := wire#w1)
      I_Contact( "Robot_Drive on status" )
      wire#w2
      Coil( "Dveře 1 otevřit" )
      Coil( "Dveře 1 otevřeno" )
   END_RUNG
   RUNG wire#powerrail
      Contact( "Dveře 1 potvrzeno zavření" )
   END_RUNG wire#w1
   RUNG wire#powerrail
      Contact( "Nouzové zastavení" )
   END_RUNG wire#w2
   // the same network as SCL:
   IF "Dveře 1 požadavek" THEN
       #"Požadavek otevření dveří 1" := TRUE;   // SR flip-flop
   END_IF;
   IF "Dveře 1 potvrzeno zavření" THEN #"Požadavek otevření dveří 1" := FALSE; END_IF;
   "Dveře 1 otevřit" := (#"Požadavek otevření dveří 1" AND NOT "Robot_Drive on status") OR "Nouzové zastavení";
   "Dveře 1 otevřeno" := "Dveře 1 otevřit";
END_REGION

REGION Network 2
   RUNG wire#powerrail
      Contact( "Dveře 2 požadavek" )
      S_SR(operand := #"Požadavek otevření dveří 2", r1 := wire#w1)
      I_Contact( "Robot_Drive on status" )
      wire#w2
      Coil( "Dveře 2 otevřit" )
      Coil( "Dveře 2 otevřeno" )
   END_RUNG
   RUNG wire#powerrail
      Contact( "Dveře 2 potvrzeno zavření" )
   END_RUNG wire#w1
   RUNG wire#powerrail
      Contact( "Nouzové zastavení" )
   END_RUNG wire#w2
   // the same network as SCL:
   IF "Dveře 2 požadavek" THEN
       #"Požadavek otevření dveří 2" := TRUE;   // SR flip-flop
   END_IF;
   IF "Dveře 2 potvrzeno zavření" THEN #"Požadavek otevření dveří 2" := FALSE; END_IF;
   "Dveře 2 otevřit" := (#"Požadavek otevření dveří 2" AND NOT "Robot_Drive on status") OR "Nouzové zastavení";
   "Dveře 2 otevřeno" := "Dveře 2 otevřit";
END_REGION
END_FUNCTION_BLOCK

FUNCTION_BLOCK "Signalni sloupek"   // FB61, LAD
{ S7_Optimized_Access := 'FALSE' }
VERSION : 0.1
BEGIN

REGION Network 1
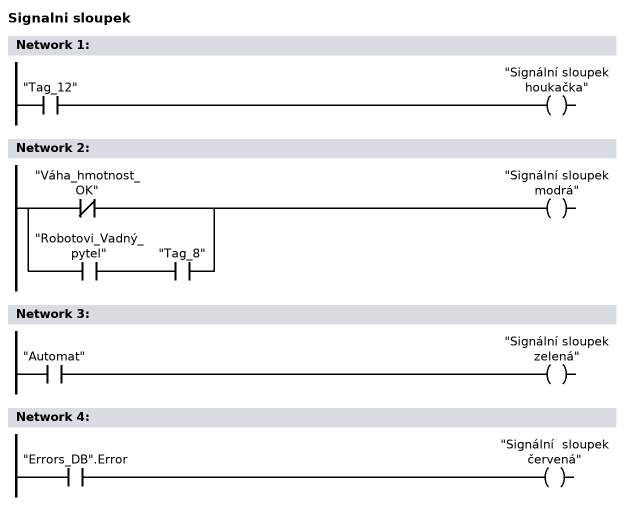
   RUNG wire#powerrail
      Contact( "Tag_12" )
      Coil( "Signální sloupek houkačka" )
   END_RUNG
   // the same network as SCL:
   "Signální sloupek houkačka" := "Tag_12";
END_REGION

REGION Network 2
   RUNG wire#powerrail
      I_Contact( "Váha_hmotnost_OK" )
      wire#w1
      Coil( "Signální sloupek modrá" )
   END_RUNG
   RUNG wire#powerrail
      Contact( "Robotovi_Vadný_pytel" )
      Contact( "Tag_8" )
   END_RUNG wire#w1
   // the same network as SCL:
   "Signální sloupek modrá" := NOT "Váha_hmotnost_OK" OR ("Robotovi_Vadný_pytel" AND "Tag_8");
END_REGION

REGION Network 3
   RUNG wire#powerrail
      Contact( "Automat" )
      Coil( "Signální sloupek zelená" )
   END_RUNG
   // the same network as SCL:
   "Signální sloupek zelená" := "Automat";
END_REGION

REGION Network 4
   RUNG wire#powerrail
      Contact( "Errors_DB".Error )
      Coil( "Signální  sloupek červená" )
   END_RUNG
   // the same network as SCL:
   "Signální  sloupek červená" := "Errors_DB".Error;
END_REGION
END_FUNCTION_BLOCK

FUNCTION_BLOCK "Errors"   // FB100, LAD
{ S7_Optimized_Access := 'FALSE' }
VERSION : 0.1
   VAR_OUTPUT
      Error : Bool;
   END_VAR
   VAR
      "Nouzové zastavení" : Bool;
      "Vypnuty silové obvody" : Bool;
      "Nízký tlak vzduchu" : Bool;
      "Jistič doptavníku P1" : Bool;
      "Jistič dopravníku P2 nebo P3" : Bool;
      "Jističe válcovačky nebo dopravníku ovíječky" : Bool;
      "Překážka ve světelné závoře" : Bool;
      "Porucha kontaktů bezpečnostního relé" : Bool;
      "Nouzové zastavení robot" : Bool;
      "Nouzové zastavení ovíječka" : Bool;
      reserva_2 : Bool;
      reserva_2_1 : Bool;
      reserva_3 : Bool;
      reserva_3_1 : Bool;
      reserva_3_2 : Bool;
      reserva_3_3 : Bool;
      "Příliš dlouhý přesun z dopravníku P2" : Bool;
      "Příliš dlouhý přesun z ovíječky" : Bool;
      "Příliš dlouhý přesun palety na dopravníku P2 ke stohu" : Bool;
      "Příliš dlouhý přesun palety na dopravníku P2 k ovíječce" : Bool;
      "Příliš dlouhý chod rovnání palety k paletě" : Bool;
      "Příliš dlouhý chod rovnání palety od palety" : Bool;
      reserve : Bool;
      reserve_1 : Bool;
      reserve_2 : Bool;
      reserve_3 : Bool;
      reserve_4 : Bool;
      reserve_5 : Bool;
      reserve_6 : Bool;
      reserve_7 : Bool;
      reserve_8 : Bool;
      reserve_9 : Bool;
   END_VAR
   VAR_TEMP   // added for the SCL form of the ladder/FBD networks
      _w1 : Bool;
      _s5time1 : S5Time;
   END_VAR
BEGIN

REGION Network 1
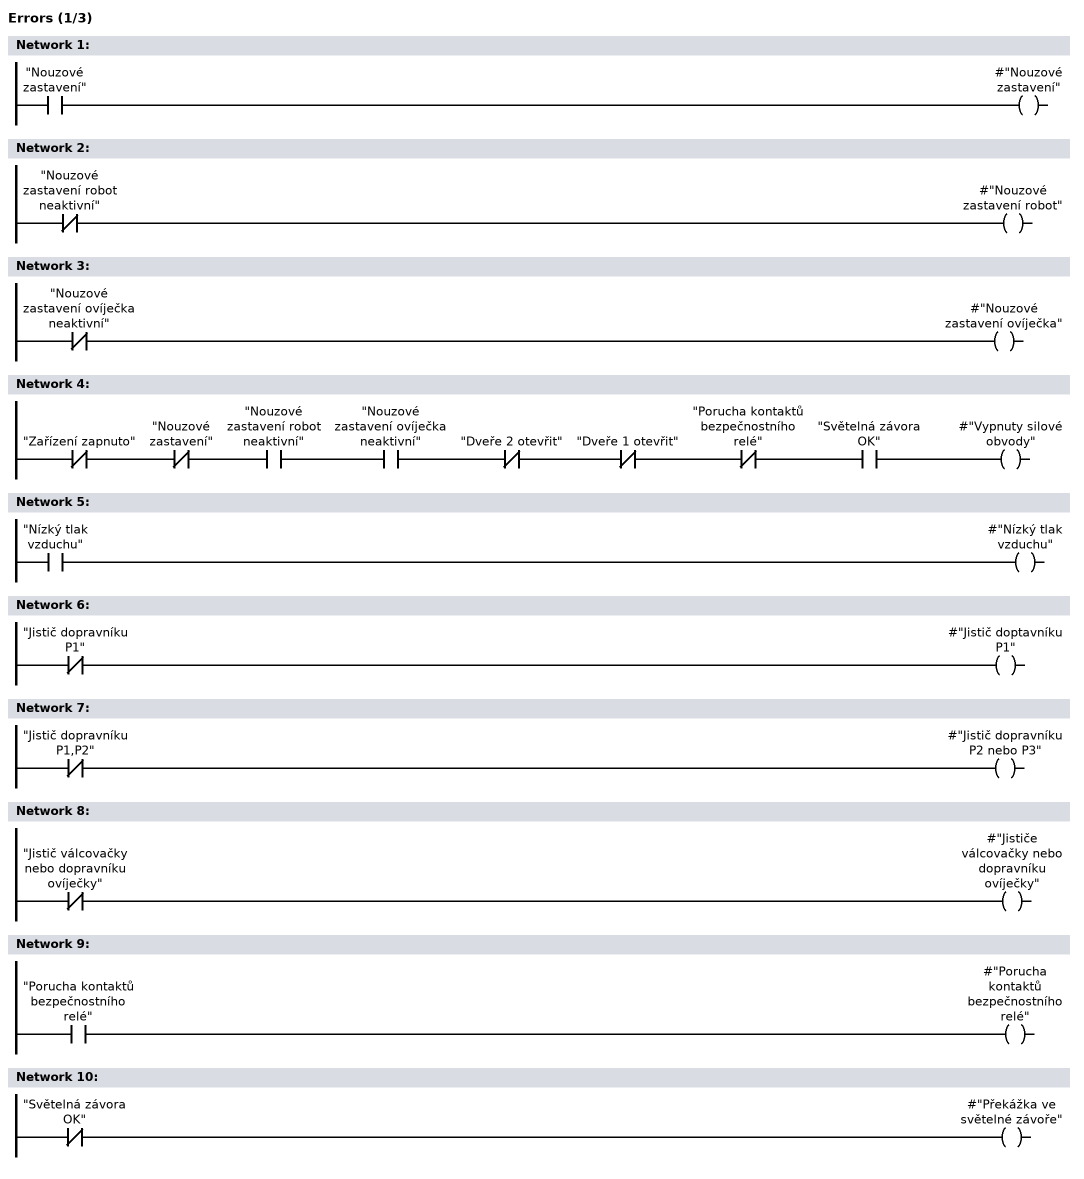
   RUNG wire#powerrail
      Contact( "Nouzové zastavení" )
      Coil( #"Nouzové zastavení" )
   END_RUNG
   // the same network as SCL:
   #"Nouzové zastavení" := "Nouzové zastavení";
END_REGION

REGION Network 2
   RUNG wire#powerrail
      I_Contact( "Nouzové zastavení robot neaktivní" )
      Coil( #"Nouzové zastavení robot" )
   END_RUNG
   // the same network as SCL:
   #"Nouzové zastavení robot" := NOT "Nouzové zastavení robot neaktivní";
END_REGION

REGION Network 3
   RUNG wire#powerrail
      I_Contact( "Nouzové zastavení ovíječka neaktivní" )
      Coil( #"Nouzové zastavení ovíječka" )
   END_RUNG
   // the same network as SCL:
   #"Nouzové zastavení ovíječka" := NOT "Nouzové zastavení ovíječka neaktivní";
END_REGION

REGION Network 4
   RUNG wire#powerrail
      I_Contact( "Zařízení zapnuto" )
      I_Contact( "Nouzové zastavení" )
      Contact( "Nouzové zastavení robot neaktivní" )
      Contact( "Nouzové zastavení ovíječka neaktivní" )
      I_Contact( "Dveře 2 otevřit" )
      I_Contact( "Dveře 1 otevřit" )
      I_Contact( "Porucha kontaktů bezpečnostního relé" )
      Contact( "Světelná závora OK" )
      Coil( #"Vypnuty silové obvody" )
   END_RUNG
   // the same network as SCL:
   #"Vypnuty silové obvody" := NOT "Zařízení zapnuto" AND NOT "Nouzové zastavení" AND "Nouzové zastavení robot neaktivní" AND "Nouzové zastavení ovíječka neaktivní" AND NOT "Dveře 2 otevřit" AND NOT "Dveře 1 otevřit" AND NOT "Porucha kontaktů bezpečnostního relé" AND "Světelná závora OK";
END_REGION

REGION Network 5
   RUNG wire#powerrail
      Contact( "Nízký tlak vzduchu" )
      Coil( #"Nízký tlak vzduchu" )
   END_RUNG
   // the same network as SCL:
   #"Nízký tlak vzduchu" := "Nízký tlak vzduchu";
END_REGION

REGION Network 6
   RUNG wire#powerrail
      I_Contact( "Jistič dopravníku P1" )
      Coil( #"Jistič doptavníku P1" )
   END_RUNG
   // the same network as SCL:
   #"Jistič doptavníku P1" := NOT "Jistič dopravníku P1";
END_REGION

REGION Network 7
   RUNG wire#powerrail
      I_Contact( "Jistič dopravníku P1,P2" )
      Coil( #"Jistič dopravníku P2 nebo P3" )
   END_RUNG
   // the same network as SCL:
   #"Jistič dopravníku P2 nebo P3" := NOT "Jistič dopravníku P1,P2";
END_REGION

REGION Network 8
   RUNG wire#powerrail
      I_Contact( "Jistič válcovačky nebo dopravníku ovíječky" )
      Coil( #"Jističe válcovačky nebo dopravníku ovíječky" )
   END_RUNG
   // the same network as SCL:
   #"Jističe válcovačky nebo dopravníku ovíječky" := NOT "Jistič válcovačky nebo dopravníku ovíječky";
END_REGION

REGION Network 9
   RUNG wire#powerrail
      Contact( "Porucha kontaktů bezpečnostního relé" )
      Coil( #"Porucha kontaktů bezpečnostního relé" )
   END_RUNG
   // the same network as SCL:
   #"Porucha kontaktů bezpečnostního relé" := "Porucha kontaktů bezpečnostního relé";
END_REGION

REGION Network 10
   RUNG wire#powerrail
      I_Contact( "Světelná závora OK" )
      Coil( #"Překážka ve světelné závoře" )
   END_RUNG
   // the same network as SCL:
   #"Překážka ve světelné závoře" := NOT "Světelná závora OK";
END_REGION

REGION Network 11
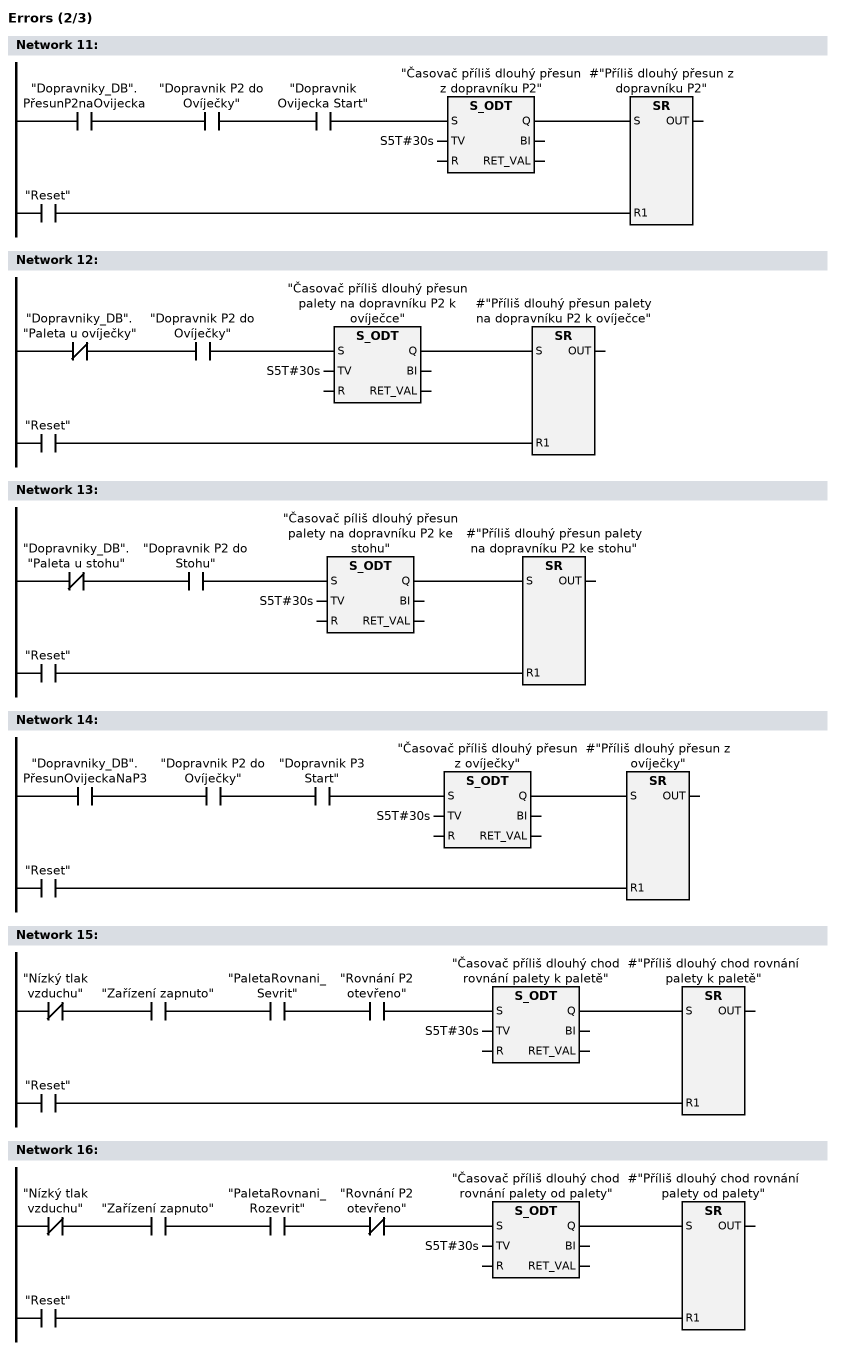
   RUNG wire#powerrail
      Contact( "Dopravniky_DB".PřesunP2naOvijecka )
      Contact( "Dopravnik P2 do Ovíječky" )
      Contact( "Dopravnik Ovijecka Start" )
      S_ODT(T_NO := "Časovač příliš dlouhý přesun z dopravníku P2", TV := S5T#30s, R :=, BI =>, RET_VAL =>)
      S_SR(operand := #"Příliš dlouhý přesun z dopravníku P2", r1 := wire#w1)
   END_RUNG
   RUNG wire#powerrail
      Contact( "Reset" )
   END_RUNG wire#w1
   // the same network as SCL:
   #_s5time1 := S_ODT(T_NO := "Časovač příliš dlouhý přesun z dopravníku P2",
                      S := "Dopravniky_DB".PřesunP2naOvijecka AND "Dopravnik P2 do Ovíječky" AND "Dopravnik Ovijecka Start",
                      TV := S5T#30s,
                      Q => #_w1);
   IF #_w1 THEN
       #"Příliš dlouhý přesun z dopravníku P2" := TRUE;   // SR flip-flop
   END_IF;
   IF "Reset" THEN #"Příliš dlouhý přesun z dopravníku P2" := FALSE; END_IF;
END_REGION

REGION Network 12
   RUNG wire#powerrail
      I_Contact( "Dopravniky_DB"."Paleta u ovíječky" )
      Contact( "Dopravnik P2 do Ovíječky" )
      S_ODT(T_NO := "Časovač příliš dlouhý přesun palety na dopravníku P2 k ovíječce", TV := S5T#30s, R :=, BI =>, RET_VAL =>)
      S_SR(operand := #"Příliš dlouhý přesun palety na dopravníku P2 k ovíječce", r1 := wire#w1)
   END_RUNG
   RUNG wire#powerrail
      Contact( "Reset" )
   END_RUNG wire#w1
   // the same network as SCL:
   #_s5time1 := S_ODT(T_NO := "Časovač příliš dlouhý přesun palety na dopravníku P2 k ovíječce",
                      S := NOT "Dopravniky_DB"."Paleta u ovíječky" AND "Dopravnik P2 do Ovíječky",
                      TV := S5T#30s,
                      Q => #_w1);
   IF #_w1 THEN
       #"Příliš dlouhý přesun palety na dopravníku P2 k ovíječce" := TRUE;   // SR flip-flop
   END_IF;
   IF "Reset" THEN #"Příliš dlouhý přesun palety na dopravníku P2 k ovíječce" := FALSE; END_IF;
END_REGION

REGION Network 13
   RUNG wire#powerrail
      I_Contact( "Dopravniky_DB"."Paleta u stohu" )
      Contact( "Dopravnik P2 do Stohu" )
      S_ODT(T_NO := "Časovač píliš dlouhý přesun palety na dopravníku P2 ke stohu", TV := S5T#30s, R :=, BI =>, RET_VAL =>)
      S_SR(operand := #"Příliš dlouhý přesun palety na dopravníku P2 ke stohu", r1 := wire#w1)
   END_RUNG
   RUNG wire#powerrail
      Contact( "Reset" )
   END_RUNG wire#w1
   // the same network as SCL:
   #_s5time1 := S_ODT(T_NO := "Časovač píliš dlouhý přesun palety na dopravníku P2 ke stohu",
                      S := NOT "Dopravniky_DB"."Paleta u stohu" AND "Dopravnik P2 do Stohu",
                      TV := S5T#30s,
                      Q => #_w1);
   IF #_w1 THEN
       #"Příliš dlouhý přesun palety na dopravníku P2 ke stohu" := TRUE;   // SR flip-flop
   END_IF;
   IF "Reset" THEN #"Příliš dlouhý přesun palety na dopravníku P2 ke stohu" := FALSE; END_IF;
END_REGION

REGION Network 14
   RUNG wire#powerrail
      Contact( "Dopravniky_DB".PřesunOvijeckaNaP3 )
      Contact( "Dopravnik P2 do Ovíječky" )
      Contact( "Dopravnik P3 Start" )
      S_ODT(T_NO := "Časovač příliš dlouhý přesun z ovíječky", TV := S5T#30s, R :=, BI =>, RET_VAL =>)
      S_SR(operand := #"Příliš dlouhý přesun z ovíječky", r1 := wire#w1)
   END_RUNG
   RUNG wire#powerrail
      Contact( "Reset" )
   END_RUNG wire#w1
   // the same network as SCL:
   #_s5time1 := S_ODT(T_NO := "Časovač příliš dlouhý přesun z ovíječky",
                      S := "Dopravniky_DB".PřesunOvijeckaNaP3 AND "Dopravnik P2 do Ovíječky" AND "Dopravnik P3 Start",
                      TV := S5T#30s,
                      Q => #_w1);
   IF #_w1 THEN
       #"Příliš dlouhý přesun z ovíječky" := TRUE;   // SR flip-flop
   END_IF;
   IF "Reset" THEN #"Příliš dlouhý přesun z ovíječky" := FALSE; END_IF;
END_REGION

REGION Network 15
   RUNG wire#powerrail
      I_Contact( "Nízký tlak vzduchu" )
      Contact( "Zařízení zapnuto" )
      Contact( "PaletaRovnani_Sevrit" )
      Contact( "Rovnání P2 otevřeno" )
      S_ODT(T_NO := "Časovač příliš dlouhý chod rovnání palety k paletě", TV := S5T#30s, R :=, BI =>, RET_VAL =>)
      S_SR(operand := #"Příliš dlouhý chod rovnání palety k paletě", r1 := wire#w1)
   END_RUNG
   RUNG wire#powerrail
      Contact( "Reset" )
   END_RUNG wire#w1
   // the same network as SCL:
   #_s5time1 := S_ODT(T_NO := "Časovač příliš dlouhý chod rovnání palety k paletě",
                      S := NOT "Nízký tlak vzduchu" AND "Zařízení zapnuto" AND "PaletaRovnani_Sevrit" AND "Rovnání P2 otevřeno",
                      TV := S5T#30s,
                      Q => #_w1);
   IF #_w1 THEN
       #"Příliš dlouhý chod rovnání palety k paletě" := TRUE;   // SR flip-flop
   END_IF;
   IF "Reset" THEN #"Příliš dlouhý chod rovnání palety k paletě" := FALSE; END_IF;
END_REGION

REGION Network 16
   RUNG wire#powerrail
      I_Contact( "Nízký tlak vzduchu" )
      Contact( "Zařízení zapnuto" )
      Contact( "PaletaRovnani_Rozevrit" )
      I_Contact( "Rovnání P2 otevřeno" )
      S_ODT(T_NO := "Časovač příliš dlouhý chod rovnání palety od palety", TV := S5T#30s, R :=, BI =>, RET_VAL =>)
      S_SR(operand := #"Příliš dlouhý chod rovnání palety od palety", r1 := wire#w1)
   END_RUNG
   RUNG wire#powerrail
      Contact( "Reset" )
   END_RUNG wire#w1
   // the same network as SCL:
   #_s5time1 := S_ODT(T_NO := "Časovač příliš dlouhý chod rovnání palety od palety",
                      S := NOT "Nízký tlak vzduchu" AND "Zařízení zapnuto" AND "PaletaRovnani_Rozevrit" AND NOT "Rovnání P2 otevřeno",
                      TV := S5T#30s,
                      Q => #_w1);
   IF #_w1 THEN
       #"Příliš dlouhý chod rovnání palety od palety" := TRUE;   // SR flip-flop
   END_IF;
   IF "Reset" THEN #"Příliš dlouhý chod rovnání palety od palety" := FALSE; END_IF;
END_REGION

REGION Network 17
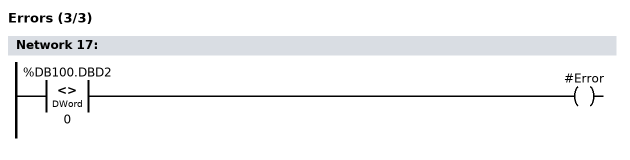
   RUNG wire#powerrail
      { S7_Templates := "SrcType := DWord" } NE_Contact(in1 := %DB100.DBD2, in2 := 0)
      Coil( #Error )
   END_RUNG
   // the same network as SCL:
   #Error := %DB100.DBD2 <> 0;
END_REGION
END_FUNCTION_BLOCK

(* ===== HMI "HMI_RT_2" =====
system functions are stored by id; their names below are inferred from use
connection "HMI_Connection_2": ETHERNET, SIMATIC S7 300/400 MPI

HMI tags "Default tag table"
   "Manual_Dopravnik_P1" : Bool = PLC Manual_Dopravnik_P1 AT %M50.1, 100 ms
   "Manual_Dopravnik_P2_k _oviječce" : Bool = PLC "Manual_Dopravnik_P2_k _oviječce" AT %M50.2, 100 ms
   "Manual_Dopravnik_P3" : Bool = PLC Manual_Dopravnik_P3 AT %M50.3, 100 ms
   "Manual_Valcovacka" : Bool = PLC Manual_Valcovacka AT %M60.5, 100 ms
   "Manual_PaletaRovnani_Rozevrit" : Bool = PLC Manual_PaletaRovnani_Rozevrit AT %M60.0, 100 ms
   "Manual_PaletaRovnani_Sevrit" : Bool = PLC Manual_PaletaRovnani_Sevrit AT %M60.2, 100 ms
   "Manual_Zarazka_P2_Dolu" : Bool = PLC Manual_Zarazka_P2_Dolu AT %M60.3, 100 ms
   "Manual_Zarazka_P2_Nahoru" : Bool = PLC Manual_Zarazka_P2_Nahoru AT %M60.4, 100 ms
   "Manual_RučníPřesunP2naOv" : Bool = PLC Manual_RučníPřesunP2naOv AT %M50.6, 1 s
   "OP_Start" : Bool = PLC OP_Start AT %M90.0, 1 s
   "Automat" : Bool = PLC Automat AT %M100.0, 1 s
   "Manual_Oviječka" : Bool = PLC Manual_Oviječka AT %M50.4, 1 s
   "Manual_Váha" : Bool = PLC Manual_Váha AT %M60.6, 1 s
   "OP_Stop" : Bool = PLC OP_Stop AT %M90.1, 1 s
   "Manual_RučníPřesunOvnaP3" : Bool = PLC Manual_RučníPřesunOvnaP3 AT %M50.5, 1 s
   "Screen" : UInt, internal
   "Errors_DB_NouzoveZastaveni" : Bool = PLC Errors_DB."Nouzové zastavení" AT %DB100.DBX2.0, 1 s
   "Manual_Paletu_P2_k_ovíječce" : Bool = PLC Manual_Paletu_P2_k_ovíječce AT %M51.1, 1 s
   "Manual_Paletu_P2_ke_stohu" : Bool = PLC Manual_Paletu_P2_ke_stohu AT %M51.0, 1 s
   "Manual_Dopravnik_P2_ke_stohu" : Bool = PLC Manual_Dopravnik_P2_ke_stohu AT %M50.7, 1 s

HMI tags "Errors"
   "Errors 1" : Int AT %DB100.DBW2, 1 s
   "Evaluated errors 1" : Int AT %DB100.DBW4, 1 s

HMI tags "Numbers"
   "Počítadlo_DB_Aktuální počet pytlů" : Int = PLC Počítadlo_DB."Aktuální počet pytlů" AT %DB5.DBW8, 1 s
   "Počítadlo_DB_Aktuální počet vrstev" : Int = PLC Počítadlo_DB."Aktuální počet vrstev" AT %DB5.DBW6, 1 s
   "Počítadlo_DB_ČísloArtiklu" : Int = PLC Počítadlo_DB.ČísloArtiklu AT %DB5.DBW0, 1 s
   "Počítadlo_DB_Počet Vrstev" : Int = PLC Počítadlo_DB."Počet Vrstev" AT %DB5.DBW4, 1 s

discrete alarms
   1: 'Central stop / Nouzové zastavení', class Chyby, trigger "Errors 1" bit 8
   2: 'Vypnuty silové obvody', class Chyby, trigger "Errors 1" bit 9
   3: 'Nízký tlak vzduchu', class Chyby, trigger "Errors 1" bit 10
   4: 'Jistič doptavníku P1', class Chyby, trigger "Errors 1" bit 11
   5: 'Jistič dopravníku P2 nebo P3', class Chyby, trigger "Errors 1" bit 12
   6: 'Jističe válcovačky nebo dopravníku ovíječky', class Chyby, trigger "Errors 1" bit 13
   7: 'reserva', class Chyby, trigger "Errors 1" bit 14
   8: 'Porucha bezpečnostního relé', class Chyby, trigger "Errors 1" bit 15
   9: 'reserva_1', class Chyby, trigger "Errors 1" bit 0
   10: 'reserva_1_1', class Chyby, trigger "Errors 1" bit 1
   11: 'reserva_2', class Chyby, trigger "Errors 1" bit 2
   12: 'reserva_2_1', class Chyby, trigger "Errors 1" bit 3
   13: 'reserva_3', class Chyby, trigger "Errors 1" bit 4
   14: 'reserva_3_1', class Chyby, trigger "Errors 1" bit 5
   15: 'reserva_3_2', class Chyby, trigger "Errors 1" bit 6
   16: 'reserva_3_3', class Chyby, trigger "Errors 1" bit 7

graphic list "Graphic_list_1": 0 'play-512'; 1 'Stop_button_play_pause_music'

screen "Root screen" 320x240, template "Template_1"
   on GenerateScreen: SetTag("Screen", 1)
   IOField "I/O field_1" at 226,123 size 30x23; FormatPattern 9
      ProcessValue <- "Počítadlo_DB_Aktuální počet pytlů"
   IOField "I/O field_2" at 226,151 size 30x23; FormatPattern 99
      ProcessValue <- "Počítadlo_DB_Aktuální počet vrstev"
   TextField "Text field_1" at 90,128 size 105x13; Text 'Aktuální počet pytlů:'
   TextField "Text field_2" at 84,156 size 112x13; Text 'Aktuální počet vrstev:'
   IOField "I/O field_3" at 226,96 size 30x23; FormatPattern 99
      ProcessValue <- "Počítadlo_DB_Počet Vrstev"
   IOField "I/O field_4" at 226,69 size 30x23; FormatPattern 99
      ProcessValue <- "Počítadlo_DB_ČísloArtiklu"
   TextField "Text field_3" at 130,74 size 65x13; Text 'Číslo artiklu:'
   TextField "Text field_4" at 78,101 size 117x13; Text 'Počet vrstev na paletě:'

screen "Manual" 320x240, template "Template_1"
   on GenerateScreen: SetTag("Screen", 2)
   Button "Button_1" at 212,40 size 96x32; TextOff 'Dopravník P1'
      on Press: SetBit("Manual_Dopravnik_P1")
      on Release: ResetBit("Manual_Dopravnik_P1")
   Button "Button_2" at 60,74 size 43x33; TextOff 'P2 ->'
      on Release: ResetBit("Manual_Dopravnik_P2_k _oviječce")
      on Press: SetBit("Manual_Dopravnik_P2_k _oviječce")
   Button "Button_3" at 212,75 size 96x32; TextOff 'Dopravník P3'
      on Release: ResetBit("Manual_Dopravnik_P3")
      on Press: SetBit("Manual_Dopravnik_P3")
   Button "Button_4" at 8,39 size 96x32; TextOff 'Válcovačka'
      on Release: ResetBit("Manual_Valcovacka")
      on Press: SetBit("Manual_Valcovacka")
   Button "Button_5" at 8,151 size 95x17; TextOff 'Rovnání sevřít'
      on Release: ResetBit("Manual_PaletaRovnani_Sevrit")
      on Press: SetBit("Manual_PaletaRovnani_Sevrit"); ResetBit("Manual_Paletu_P2_k_ovíječce"); ResetBit("Manual_Paletu_P2_ke_stohu")
   Button "Button_6" at 8,181 size 95x17; TextOff 'Rovnání rozevřít'
      on Release: ResetBit("Manual_PaletaRovnani_Rozevrit")
      on Press: SetBit("Manual_PaletaRovnani_Rozevrit"); ResetBit("Manual_Paletu_P2_k_ovíječce"); ResetBit("Manual_Paletu_P2_ke_stohu")
   Button "Button_7" at 116,157 size 96x32; TextOff 'Paleta ke stohu'
      on Press: SetBit("Manual_Paletu_P2_ke_stohu"); ResetBit("Manual_Paletu_P2_k_ovíječce")
   Button "Button_8" at 214,157 size 94x32; TextOff 'Paleta k ovíječce'
      on Press: SetBit("Manual_Paletu_P2_k_ovíječce"); ResetBit("Manual_Paletu_P2_ke_stohu")
   Button "Button_9" at 111,75 size 96x32; TextOff 'Ovíječka'
      on Release: ResetBit("Manual_Oviječka")
      on Press: SetBit("Manual_Oviječka")
   Button "Button_10" at 111,39 size 96x32; TextOff 'Váha'
      on Release: ResetBit("Manual_Váha")
      on Press: SetBit("Manual_Váha")
   Button "Button_11" at 58,112 size 96x32; TextOff 'P2 na Ov'
      on Release: ResetBit("Manual_RučníPřesunP2naOv")
      on Press: SetBit("Manual_RučníPřesunP2naOv")
   Button "Button_12" at 164,112 size 96x32; TextOff 'Ov na P3'
      on Release: ResetBit("Manual_RučníPřesunOvnaP3")
      on Press: SetBit("Manual_RučníPřesunOvnaP3")
   Button "Button_13" at 8,74 size 43x32; TextOff '<- P2'
      on Release: ResetBit("Manual_Dopravnik_P2_ke_stohu")
      on Press: SetBit("Manual_Dopravnik_P2_ke_stohu")

screen "Setting" 320x240, template "Template_1"
   on GenerateScreen: SetTag("Screen", 3)
   Button "Button_1" at 25,60 size 75x28; TextOff 'Login / Přihlášení'
      on Press: function_a2a04561()
   Button "Button_2" at 25,105 size 75x28; TextOff 'Logout / Odhlášení'
      on Press: function_f23ef4c9()
   Button "Button_3" at 165,60 size 96x32; TextOff 'Text'
      on Release: function_ef3f5d25("Alarm window_Unacknowledged", -1)

Template "Template_1" 320x240
   Button "Exit" at 266,202 size 52x37; TextOff 'Exit'; PictureOff "ExitRuntime_KTP600_Basic_color_PN"; PictureOn "ExitRuntime_KTP600_Basic_color_PN"; Authorization "User administration"
      on Release: StopRuntime(0)
   Button "Template_Button" at 213,202 size 52x37; TextOff 'Text'; PictureOff "custom_settings-512"
      on Release: ActivateScreen("Setting", 0)
   Button "Template_Button_1" at 160,202 size 52x37; TextOff 'Text'; PictureOff "Hand-Touch-icon-300x300"
      on Release: ActivateScreen("Manual", 0)
   Button "Template_Button_2" at 107,202 size 52x37; TextOff 'Text'; PictureList "Graphic_list_1"
      ProcessValue <- "Automat"
      on Press: SetBit("OP_Start")
      on Release: ResetBit("OP_Start")
   Button "Alarms" at 54,202 size 52x37; TextOff 'Alarms'; PictureOff "AlarmDisplay_KTP600_Basic_color_PN"; PictureOn "AlarmDisplay_KTP600_Basic_color_PN"
      on Release: ActivateScreen("Alarms", 0)
   Button "Start screen" at 1,202 size 52x37; TextOff 'Start screen'; PictureOff "NavigateHome_KTP600_Basic_color_PN"; PictureOn "NavigateHome_KTP600_Basic_color_PN"
      on Release: ActivateScreen("Root screen", 0)
   DateTimeField "HmiScreenItemData" at 235,19 size 85x19
   DateTimeField "HmiScreenItemData_1" at 235,0 size 85x19
   GraphicView "Logo" at 8,11 size 125x22; Picture "logo"

screen "Alarms" 320x240, template "Template_1"
   AlarmView "Alarm view_1" at 0,41 size 320x151
*)